LIN {X 0,Y 176.78,Z 239.076,A -85,B 0,C 180,E1 -23448.194,E2 -23448.194} C_VEL
LIN {X 0,Y 178.363,Z 246.541,A -85,B 0,C 180,E1 -23449.914,E2 -23449.914} C_VEL
LIN {X 0,Y 179.453,Z 256.138,A -85,B 0,C 180,E1 -23452.116,E2 -23452.116} C_VEL
LIN {X 0,Y 179.616,Z 266.645,A -85,B 0,C 180,E1 -23454.675,E2 -23454.675} C_VEL
LIN {X 0,Y 179.07,Z 275.287,A -85,B 0,C 180,E1 -23457.005,E2 -23457.005} C_VEL
LIN {X 0,Y 178.404,Z 280.467,A -85,B 0,C 180,E1 -23458.535,E2 -23458.535} C_VEL
LIN {X 0,Y 175.026,Z 289.302,A -85,B 0,C 180,E1 -23461.193,E2 -23461.193} C_VEL
LIN {X 0,Y 171.949,Z 296.845,A -85,B 0,C 180,E1 -23464.053,E2 -23464.053} C_VEL
LIN {X 0,Y 168.882,Z 303.785,A -85,B 0,C 180,E1 -23467.36,E2 -23467.36} C_VEL
LIN {X 0,Y 166.698,Z 308.639,A -85,B 0,C 180,E1 -23470.288,E2 -23470.288} C_VEL
LIN {X 0,Y 164.538,Z 313.357,A -85,B 0,C 180,E1 -23473.88,E2 -23473.88} C_VEL
LIN {X 0,Y 163.144,Z 316.97,A -85,B 0,C 180,E1 -23477.561,E2 -23477.561} C_VEL
LIN {X 0,Y 162.461,Z 318.833,A -85,B 0,C 180,E1 -23480.035,E2 -23480.035} C_VEL
LIN {X 0,Y 161.851,Z 321.235,A -85,B 0,C 180,E1 -23485.017,E2 -23485.017} C_VEL
LIN {X 0,Y 161.779,Z 321.876,A -85,B 0,C 180,E1 -23487.66,E2 -23487.66} C_VEL
LIN {X 0,Y 161.892,Z 322.064,A -85,B 0,C 180,E1 -23489.999,E2 -23489.999} C_VEL
LIN {X 0,Y 161.797,Z 321.836,A -85,B 0,C 180,E1 -23492.489,E2 -23492.489} C_VEL
LIN {X 0,Y 161.851,Z 321.217,A -85,B 0,C 180,E1 -23494.982,E2 -23494.982} C_VEL
LIN {X 0,Y 162.035,Z 320.208,A -85,B 0,C 180,E1 -23497.476,E2 -23497.476} C_VEL
LIN {X 0,Y 162.46,Z 318.797,A -85,B 0,C 180,E1 -23499.964,E2 -23499.964} C_VEL
LIN {X 0,Y 163.562,Z 315.842,A -85,B 0,C 180,E1 -23503.669,E2 -23503.669} C_VEL
LIN {X 0,Y 165.153,Z 311.848,A -85,B 0,C 180,E1 -23507.33,E2 -23507.33} C_VEL
LIN {X 0,Y 167.973,Z 305.719,A -85,B 0,C 180,E1 -23511.475,E2 -23511.475} C_VEL
LIN {X 0,Y 170.948,Z 299.153,A -85,B 0,C 180,E1 -23514.858,E2 -23514.858} C_VEL
LIN {X 0,Y 173.284,Z 293.389,A -85,B 0,C 180,E1 -23517.287,E2 -23517.287} C_VEL
LIN {X 0,Y 174.194,Z 289.612,A -85,B 0,C 180,E1 -23518.754,E2 -23518.754} C_VEL
LIN {X 0,Y 174.206,Z 285.779,A -85,B 0,C 180,E1 -23520.268,E2 -23520.268} C_VEL
LIN {X 0,Y 173.026,Z 275.11,A -85,B 0,C 180,E1 -23524.233,E2 -23524.233} C_VEL
LIN {X 0,Y 173.101,Z 272.13,A -85,B 0,C 180,E1 -23525.13,E2 -23525.13} C_VEL
LIN {X 0,Y 173.392,Z 261.231,A -85,B 0,C 180,E1 -23528.088,E2 -23528.088} C_VEL
LIN {X 0,Y 172.773,Z 251.105,A -85,B 0,C 180,E1 -23530.604,E2 -23530.604} C_VEL
LIN {X 0,Y 171.555,Z 243.424,A -85,B 0,C 180,E1 -23532.49,E2 -23532.49} C_VEL
LIN {X 0,Y 169.435,Z 236.666,A -85,B 0,C 180,E1 -23534.315,E2 -23534.315} C_VEL
LIN {X 0,Y 166.079,Z 229.215,A -85,B 0,C 180,E1 -23536.586,E2 -23536.586} C_VEL
LIN {X 0,Y 163.832,Z 224.747,A -85,B 0,C 180,E1 -23538.015,E2 -23538.015} C_VEL
LIN {X 0,Y 161.816,Z 220.984,A -85,B 0,C 180,E1 -23539.276,E2 -23539.276} C_VEL
LIN {X 0,Y 160.918,Z 219.536,A -85,B 0,C 180,E1 -23539.797,E2 -23539.797} C_VEL
LIN {X 0,Y 158.85,Z 216.171,A -85,B 0,C 180,E1 -23541.045,E2 -23541.045} C_VEL
LIN {X 0,Y 158.329,Z 214.418,A -85,B 0,C 180,E1 -23541.503,E2 -23541.503} C_VEL
LIN {X 0,Y 158.132,Z 212.84,A -85,B 0,C 180,E1 -23544.706,E2 -23544.706} C_VEL
LIN {X 0,Y 157.933,Z 211.437,A -85,B 0,C 180,E1 -23547.724,E2 -23547.724} C_VEL
LIN {X 0,Y 157.54,Z 209.207,A -85,B 0,C 180,E1 -23553.151,E2 -23553.151} C_VEL
LIN {X 0,Y 157.335,Z 208.061,A -85,B 0,C 180,E1 -23556.295,E2 -23556.295} C_VEL
LIN {X 0,Y 157.408,Z 207.878,A -85,B 0,C 180,E1 -23561.788,E2 -23561.788} C_VEL
LIN {X 0,Y 157.528,Z 207.864,A -85,B 0,C 180,E1 -23567.111,E2 -23567.111} C_VEL
LIN {X 0,Y 157.685,Z 207.834,A -85,B 0,C 180,E1 -23569.731,E2 -23569.731} C_VEL
LIN {X 0,Y 157.759,Z 207.833,A -85,B 0,C 180,E1 -23572.32,E2 -23572.32} C_VEL
LIN {X 0,Y 158.255,Z 207.772,A -85,B 0,C 180,E1 -23580,E2 -23580} C_VEL
LIN {X 0,Y 157.76,Z 207.832,A -85,B 0,C 180,E1 -23587.68,E2 -23587.68} C_VEL
LIN {X 0,Y 157.635,Z 207.85,A -85,B 0,C 180,E1 -23591.236,E2 -23591.236} C_VEL
LIN {X 0,Y 157.441,Z 207.871,A -85,B 0,C 180,E1 -23595.536,E2 -23595.536} C_VEL
LIN {X 0,Y 157.369,Z 207.88,A -85,B 0,C 180,E1 -23600.933,E2 -23600.933} C_VEL
LIN {X 0,Y 157.314,Z 207.89,A -85,B 0,C 180,E1 -23606.686,E2 -23606.686} C_VEL
LIN {X 0,Y 157.274,Z 207.896,A -85,B 0,C 180,E1 -23612.428,E2 -23612.428} C_VEL
LIN {X 0,Y 157.286,Z 207.969,A -85,B 0,C 180,E1 -23615.513,E2 -23615.513} C_VEL
LIN {X 0,Y 157.382,Z 209.037,A -85,B 0,C 180,E1 -23618.22,E2 -23618.22} C_VEL
LIN {X 0,Y 158.609,Z 211.909,A -85,B 0,C 180,E1 -23619.089,E2 -23619.089} C_VEL
LIN {X 0,Y 160.841,Z 214.656,A -85,B 0,C 180,E1 -23620.365,E2 -23620.365} C_VEL
LIN {X 0,Y 162.87,Z 218.288,A -85,B 0,C 180,E1 -23621.667,E2 -23621.667} C_VEL
LIN {X 0,Y 164.29,Z 220.876,A -85,B 0,C 180,E1 -23622.565,E2 -23622.565} C_VEL
LIN {X 0,Y 166.657,Z 225.258,A -85,B 0,C 180,E1 -23624.094,E2 -23624.094} C_VEL
LIN {X 0,Y 170.357,Z 233.531,A -85,B 0,C 180,E1 -23626.764,E2 -23626.764} C_VEL
LIN {X 0,Y 172.946,Z 242.042,A -85,B 0,C 180,E1 -23629.234,E2 -23629.234} C_VEL
LIN {X 0,Y 174.494,Z 250.978,A -85,B 0,C 180,E1 -23631.721,E2 -23631.721} C_VEL
LIN {X 0,Y 175.228,Z 260.194,A -85,B 0,C 180,E1 -23634.39,E2 -23634.39} C_VEL
LIN {X 0,Y 175.165,Z 267.085,A -85,B 0,C 180,E1 -23636.518,E2 -23636.518} C_VEL
LIN {X 0,Y 171.645,Z 276.507,A -85,B 0,C 180,E1 -23639.153,E2 -23639.153} C_VEL
LIN {X 0,Y 168.395,Z 284.517,A -85,B 0,C 180,E1 -23641.998,E2 -23641.998} C_VEL
LIN {X 0,Y 164.708,Z 292.19,A -85,B 0,C 180,E1 -23645.417,E2 -23645.417} C_VEL
LIN {X 0,Y 161.162,Z 299.236,A -85,B 0,C 180,E1 -23649.583,E2 -23649.583} C_VEL
LIN {X 0,Y 158.79,Z 303.922,A -85,B 0,C 180,E1 -23653.281,E2 -23653.281} C_VEL
LIN {X 0,Y 157.051,Z 307.504,A -85,B 0,C 180,E1 -23657.071,E2 -23657.071} C_VEL
LIN {X 0,Y 156.173,Z 309.352,A -85,B 0,C 180,E1 -23659.631,E2 -23659.631} C_VEL
LIN {X 0,Y 155.582,Z 310.738,A -85,B 0,C 180,E1 -23662.212,E2 -23662.212} C_VEL
LIN {X 0,Y 154.905,Z 312.331,A -85,B 0,C 180,E1 -23667.4,E2 -23667.4} C_VEL
LIN {X 0,Y 154.88,Z 312.556,A -85,B 0,C 180,E1 -23670.001,E2 -23670.001} C_VEL
LIN {X 0,Y 154.976,Z 312.124,A -85,B 0,C 180,E1 -23673.9,E2 -23673.9} C_VEL
LIN {X 0,Y 155.582,Z 310.806,A -85,B 0,C 180,E1 -23677.789,E2 -23677.789} C_VEL
LIN {X 0,Y 156.167,Z 309.45,A -85,B 0,C 180,E1 -23680.371,E2 -23680.371} C_VEL
LIN {X 0,Y 157.516,Z 306.582,A -85,B 0,C 180,E1 -23684.206,E2 -23684.206} C_VEL
LIN {X 0,Y 159.47,Z 302.69,A -85,B 0,C 180,E1 -23687.969,E2 -23687.969} C_VEL
LIN {X 0,Y 162.031,Z 297.666,A -85,B 0,C 180,E1 -23691.635,E2 -23691.635} C_VEL
LIN {X 0,Y 165.215,Z 291.334,A -85,B 0,C 180,E1 -23695.176,E2 -23695.176} C_VEL
LIN {X 0,Y 168.946,Z 283.412,A -85,B 0,C 180,E1 -23698.581,E2 -23698.581} C_VEL
LIN {X 0,Y 172.13,Z 275.519,A -85,B 0,C 180,E1 -23701.303,E2 -23701.303} C_VEL
LIN {X 0,Y 175.172,Z 267.617,A -85,B 0,C 180,E1 -23703.481,E2 -23703.481} C_VEL
LIN {X 0,Y 175.196,Z 258.051,A -85,B 0,C 180,E1 -23706.396,E2 -23706.396} C_VEL
LIN {X 0,Y 174.062,Z 247.419,A -85,B 0,C 180,E1 -23709.43,E2 -23709.43} C_VEL
LIN {X 0,Y 172.145,Z 238.94,A -85,B 0,C 180,E1 -23711.833,E2 -23711.833} C_VEL
LIN {X 0,Y 169.321,Z 230.807,A -85,B 0,C 180,E1 -23714.275,E2 -23714.275} C_VEL
LIN {X 0,Y 165.276,Z 222.609,A -85,B 0,C 180,E1 -23717.013,E2 -23717.013} C_VEL
LIN {X 0,Y 162.881,Z 218.324,A -85,B 0,C 180,E1 -23718.543,E2 -23718.543} C_VEL
LIN {X 0,Y 160.997,Z 214.957,A -85,B 0,C 180,E1 -23719.76,E2 -23719.76} C_VEL
LIN {X 0,Y 160.149,Z 213.715,A -85,B 0,C 180,E1 -23720.261,E2 -23720.261} C_VEL
LIN {X 0,Y 157.986,Z 210.749,A -85,B 0,C 180,E1 -23721.558,E2 -23721.558} C_VEL
LIN {X 0,Y 157.382,Z 208.874,A -85,B 0,C 180,E1 -23722.095,E2 -23722.095} C_VEL
LIN {X 0,Y 157.303,Z 208.062,A -85,B 0,C 180,E1 -23724.492,E2 -23724.492} C_VEL
LIN {X 0,Y 157.294,Z 207.888,A -85,B 0,C 180,E1 -23728.096,E2 -23728.096} C_VEL
LIN {X 0,Y 157.323,Z 207.883,A -85,B 0,C 180,E1 -23733.466,E2 -23733.466} C_VEL
LIN {X 0,Y 157.396,Z 207.879,A -85,B 0,C 180,E1 -23739.667,E2 -23739.667} C_VEL
LIN {X 0,Y 157.456,Z 207.872,A -85,B 0,C 180,E1 -23744.466,E2 -23744.466} C_VEL
LIN {X 0,Y 157.689,Z 207.842,A -85,B 0,C 180,E1 -23749.731,E2 -23749.731} C_VEL
LIN {X 0,Y 157.763,Z 207.832,A -85,B 0,C 180,E1 -23752.32,E2 -23752.32} C_VEL
LIN {X 0,Y 158.258,Z 207.77,A -85,B 0,C 180,E1 -23760,E2 -23760} C_VEL
LIN {X 0,Y 157.762,Z 207.834,A -85,B 0,C 180,E1 -23767.68,E2 -23767.68} C_VEL
LIN {X 0,Y 157.638,Z 207.852,A -85,B 0,C 180,E1 -23771.236,E2 -23771.236} C_VEL
LIN {X 0,Y 157.456,Z 207.875,A -85,B 0,C 180,E1 -23775.534,E2 -23775.534} C_VEL
LIN {X 0,Y 157.369,Z 207.883,A -85,B 0,C 180,E1 -23780.933,E2 -23780.933} C_VEL
LIN {X 0,Y 157.345,Z 208.125,A -85,B 0,C 180,E1 -23783.703,E2 -23783.703} C_VEL
LIN {X 0,Y 157.737,Z 210.255,A -85,B 0,C 180,E1 -23789.347,E2 -23789.347} C_VEL
LIN {X 0,Y 157.936,Z 211.5,A -85,B 0,C 180,E1 -23792.275,E2 -23792.275} C_VEL
LIN {X 0,Y 158.257,Z 213.7,A -85,B 0,C 180,E1 -23796.93,E2 -23796.93} C_VEL
LIN {X 0,Y 158.366,Z 214.446,A -85,B 0,C 180,E1 -23798.411,E2 -23798.411} C_VEL
LIN {X 0,Y 159.443,Z 217.379,A -85,B 0,C 180,E1 -23799.216,E2 -23799.216} C_VEL
LIN {X 0,Y 161.67,Z 220.578,A -85,B 0,C 180,E1 -23800.499,E2 -23800.499} C_VEL
LIN {X 0,Y 163.729,Z 224.606,A -85,B 0,C 180,E1 -23801.811,E2 -23801.811} C_VEL
LIN {X 0,Y 164.856,Z 226.613,A -85,B 0,C 180,E1 -23802.488,E2 -23802.488} C_VEL
LIN {X 0,Y 168.352,Z 233.944,A -85,B 0,C 180,E1 -23804.791,E2 -23804.791} C_VEL
LIN {X 0,Y 170.991,Z 241.181,A -85,B 0,C 180,E1 -23806.849,E2 -23806.849} C_VEL
LIN {X 0,Y 172.408,Z 247.523,A -85,B 0,C 180,E1 -23808.463,E2 -23808.463} C_VEL
LIN {X 0,Y 173.47,Z 258.738,A -85,B 0,C 180,E1 -23811.221,E2 -23811.221} C_VEL
LIN {X 0,Y 173.357,Z 268.826,A -85,B 0,C 180,E1 -23813.862,E2 -23813.862} C_VEL
LIN {X 0,Y 172.45,Z 278.275,A -85,B 0,C 180,E1 -23816.62,E2 -23816.62} C_VEL
LIN {X 0,Y 171.68,Z 282.204,A -85,B 0,C 180,E1 -23817.847,E2 -23817.847} C_VEL
LIN {X 0,Y 168.134,Z 290.669,A -85,B 0,C 180,E1 -23820.583,E2 -23820.583} C_VEL
LIN {X 0,Y 164.781,Z 298.441,A -85,B 0,C 180,E1 -23823.8,E2 -23823.8} C_VEL
LIN {X 0,Y 161.332,Z 305.608,A -85,B 0,C 180,E1 -23827.593,E2 -23827.593} C_VEL
LIN {X 0,Y 158.373,Z 311.709,A -85,B 0,C 180,E1 -23831.902,E2 -23831.902} C_VEL
LIN {X 0,Y 156.631,Z 315.682,A -85,B 0,C 180,E1 -23835.712,E2 -23835.712} C_VEL
LIN {X 0,Y 155.457,Z 318.62,A -85,B 0,C 180,E1 -23839.581,E2 -23839.581} C_VEL
LIN {X 0,Y 154.757,Z 321.022,A -85,B 0,C 180,E1 -23844.788,E2 -23844.788} C_VEL
LIN {X 0,Y 154.686,Z 321.748,A -85,B 0,C 180,E1 -23848.284,E2 -23848.284} C_VEL
LIN {X 0,Y 154.794,Z 321.851,A -85,B 0,C 180,E1 -23849.999,E2 -23849.999} C_VEL
LIN {X 0,Y 154.699,Z 321.623,A -85,B 0,C 180,E1 -23852.603,E2 -23852.603} C_VEL
LIN {X 0,Y 154.757,Z 321.003,A -85,B 0,C 180,E1 -23855.21,E2 -23855.21} C_VEL
LIN {X 0,Y 154.98,Z 319.994,A -85,B 0,C 180,E1 -23857.818,E2 -23857.818} C_VEL
LIN {X 0,Y 155.457,Z 318.583,A -85,B 0,C 180,E1 -23860.418,E2 -23860.418} C_VEL
LIN {X 0,Y 156.63,Z 315.627,A -85,B 0,C 180,E1 -23864.287,E2 -23864.287} C_VEL
LIN {X 0,Y 158.371,Z 311.633,A -85,B 0,C 180,E1 -23868.097,E2 -23868.097} C_VEL
LIN {X 0,Y 161.326,Z 305.502,A -85,B 0,C 180,E1 -23872.406,E2 -23872.406} C_VEL
LIN {X 0,Y 164.723,Z 298.399,A -85,B 0,C 180,E1 -23876.159,E2 -23876.159} C_VEL
LIN {X 0,Y 168.12,Z 290.511,A -85,B 0,C 180,E1 -23879.418,E2 -23879.418} C_VEL
LIN {X 0,Y 171.652,Z 282.002,A -85,B 0,C 180,E1 -23882.158,E2 -23882.158} C_VEL
LIN {X 0,Y 172.948,Z 273.749,A -85,B 0,C 180,E1 -23884.674,E2 -23884.674} C_VEL
LIN {X 0,Y 173.101,Z 272.13,A -85,B 0,C 180,E1 -23885.13,E2 -23885.13} C_VEL
LIN {X 0,Y 172.797,Z 267.849,A -85,B 0,C 180,E1 -23886.461,E2 -23886.461} C_VEL
LIN {X 0,Y 171.547,Z 263.857,A -85,B 0,C 180,E1 -23887.875,E2 -23887.875} C_VEL
LIN {X 0,Y 168.128,Z 256.123,A -85,B 0,C 180,E1 -23890.762,E2 -23890.762} C_VEL
LIN {X 0,Y 166.649,Z 250.286,A -85,B 0,C 180,E1 -23892.564,E2 -23892.564} C_VEL
LIN {X 0,Y 165.32,Z 243.61,A -85,B 0,C 180,E1 -23894.412,E2 -23894.412} C_VEL
LIN {X 0,Y 163.024,Z 237.373,A -85,B 0,C 180,E1 -23896.389,E2 -23896.389} C_VEL
LIN {X 0,Y 159.703,Z 229.94,A -85,B 0,C 180,E1 -23898.902,E2 -23898.902} C_VEL
LIN {X 0,Y 157.677,Z 225.941,A -85,B 0,C 180,E1 -23900.362,E2 -23900.362} C_VEL
LIN {X 0,Y 154.955,Z 221.098,A -85,B 0,C 180,E1 -23902.26,E2 -23902.26} C_VEL
LIN {X 0,Y 154.306,Z 219.798,A -85,B 0,C 180,E1 -23902.726,E2 -23902.726} C_VEL
LIN {X 0,Y 151.874,Z 216.371,A -85,B 0,C 180,E1 -23904.354,E2 -23904.354} C_VEL
LIN {X 0,Y 151.145,Z 214.074,A -85,B 0,C 180,E1 -23905.074,E2 -23905.074} C_VEL
LIN {X 0,Y 150.856,Z 212.313,A -85,B 0,C 180,E1 -23909.172,E2 -23909.172} C_VEL
LIN {X 0,Y 150.639,Z 211.045,A -85,B 0,C 180,E1 -23912.427,E2 -23912.427} C_VEL
LIN {X 0,Y 150.334,Z 209.112,A -85,B 0,C 180,E1 -23918.038,E2 -23918.038} C_VEL
LIN {X 0,Y 150.348,Z 208.759,A -85,B 0,C 180,E1 -23919.209,E2 -23919.209} C_VEL
LIN {X 0,Y 150.36,Z 208.755,A -85,B 0,C 180,E1 -23923.713,E2 -23923.713} C_VEL
LIN {X 0,Y 150.608,Z 208.714,A -85,B 0,C 180,E1 -23929.242,E2 -23929.242} C_VEL
LIN {X 0,Y 150.697,Z 208.714,A -85,B 0,C 180,E1 -23931.957,E2 -23931.957} C_VEL
LIN {X 0,Y 151.215,Z 208.65,A -85,B 0,C 180,E1 -23940,E2 -23940} C_VEL
LIN {X 0,Y 150.698,Z 208.713,A -85,B 0,C 180,E1 -23948.043,E2 -23948.043} C_VEL
LIN {X 0,Y 150.575,Z 208.729,A -85,B 0,C 180,E1 -23951.436,E2 -23951.436} C_VEL
LIN {X 0,Y 150.353,Z 208.755,A -85,B 0,C 180,E1 -23956.288,E2 -23956.288} C_VEL
LIN {X 0,Y 150.35,Z 208.754,A -85,B 0,C 180,E1 -23960.793,E2 -23960.793} C_VEL
LIN {X 0,Y 150.244,Z 208.769,A -85,B 0,C 180,E1 -23967.283,E2 -23967.283} C_VEL
LIN {X 0,Y 150.214,Z 208.775,A -85,B 0,C 180,E1 -23972.633,E2 -23972.633} C_VEL
LIN {X 0,Y 150.293,Z 209.416,A -85,B 0,C 180,E1 -23974.643,E2 -23974.643} C_VEL
LIN {X 0,Y 151.514,Z 212.159,A -85,B 0,C 180,E1 -23975.642,E2 -23975.642} C_VEL
LIN {X 0,Y 153.905,Z 215.12,A -85,B 0,C 180,E1 -23977.237,E2 -23977.237} C_VEL
LIN {X 0,Y 155.901,Z 218.643,A -85,B 0,C 180,E1 -23978.703,E2 -23978.703} C_VEL
LIN {X 0,Y 157.105,Z 220.386,A -85,B 0,C 180,E1 -23979.5,E2 -23979.5} C_VEL
LIN {X 0,Y 161.042,Z 227.816,A -85,B 0,C 180,E1 -23982.396,E2 -23982.396} C_VEL
LIN {X 0,Y 164.498,Z 235.616,A -85,B 0,C 180,E1 -23985.168,E2 -23985.168} C_VEL
LIN {X 0,Y 166.874,Z 243.25,A -85,B 0,C 180,E1 -23987.636,E2 -23987.636} C_VEL
LIN {X 0,Y 168.41,Z 252.094,A -85,B 0,C 180,E1 -23990.307,E2 -23990.307} C_VEL
LIN {X 0,Y 169.014,Z 261.573,A -85,B 0,C 180,E1 -23993.23,E2 -23993.23} C_VEL
LIN {X 0,Y 168.883,Z 268.368,A -85,B 0,C 180,E1 -23995.46,E2 -23995.46} C_VEL
LIN {X 0,Y 165.511,Z 276.891,A -85,B 0,C 180,E1 -23997.944,E2 -23997.944} C_VEL
LIN {X 0,Y 162.157,Z 284.733,A -85,B 0,C 180,E1 -24000.819,E2 -24000.819} C_VEL
LIN {X 0,Y 158.289,Z 292.405,A -85,B 0,C 180,E1 -24004.349,E2 -24004.349} C_VEL
LIN {X 0,Y 154.513,Z 299.451,A -85,B 0,C 180,E1 -24008.662,E2 -24008.662} C_VEL
LIN {X 0,Y 152.007,Z 304.137,A -85,B 0,C 180,E1 -24012.512,E2 -24012.512} C_VEL
LIN {X 0,Y 150.143,Z 307.718,A -85,B 0,C 180,E1 -24016.465,E2 -24016.465} C_VEL
LIN {X 0,Y 149.185,Z 309.567,A -85,B 0,C 180,E1 -24019.139,E2 -24019.139} C_VEL
LIN {X 0,Y 148.546,Z 310.952,A -85,B 0,C 180,E1 -24021.841,E2 -24021.841} C_VEL
LIN {X 0,Y 147.825,Z 312.544,A -85,B 0,C 180,E1 -24027.276,E2 -24027.276} C_VEL
LIN {X 0,Y 147.782,Z 312.769,A -85,B 0,C 180,E1 -24030.001,E2 -24030.001} C_VEL
LIN {X 0,Y 147.84,Z 312.467,A -85,B 0,C 180,E1 -24033.338,E2 -24033.338} C_VEL
LIN {X 0,Y 148.546,Z 311.019,A -85,B 0,C 180,E1 -24038.161,E2 -24038.161} C_VEL
LIN {X 0,Y 149.178,Z 309.663,A -85,B 0,C 180,E1 -24040.863,E2 -24040.863} C_VEL
LIN {X 0,Y 150.637,Z 306.795,A -85,B 0,C 180,E1 -24044.869,E2 -24044.869} C_VEL
LIN {X 0,Y 152.737,Z 302.902,A -85,B 0,C 180,E1 -24048.79,E2 -24048.79} C_VEL
LIN {X 0,Y 155.455,Z 297.878,A -85,B 0,C 180,E1 -24052.599,E2 -24052.599} C_VEL
LIN {X 0,Y 158.826,Z 291.545,A -85,B 0,C 180,E1 -24056.264,E2 -24056.264} C_VEL
LIN {X 0,Y 162.722,Z 283.659,A -85,B 0,C 180,E1 -24059.764,E2 -24059.764} C_VEL
LIN {X 0,Y 166.108,Z 275.729,A -85,B 0,C 180,E1 -24062.575,E2 -24062.575} C_VEL
LIN {X 0,Y 168.886,Z 268.892,A -85,B 0,C 180,E1 -24064.541,E2 -24064.541} C_VEL
LIN {X 0,Y 169.099,Z 260.842,A -85,B 0,C 180,E1 -24067.168,E2 -24067.168} C_VEL
LIN {X 0,Y 168.327,Z 250.867,A -85,B 0,C 180,E1 -24070.238,E2 -24070.238} C_VEL
LIN {X 0,Y 166.903,Z 243.346,A -85,B 0,C 180,E1 -24072.53,E2 -24072.53} C_VEL
LIN {X 0,Y 164.206,Z 234.837,A -85,B 0,C 180,E1 -24075.296,E2 -24075.296} C_VEL
LIN {X 0,Y 160.835,Z 227.437,A -85,B 0,C 180,E1 -24077.975,E2 -24077.975} C_VEL
LIN {X 0,Y 158.51,Z 223.061,A -85,B 0,C 180,E1 -24079.68,E2 -24079.68} C_VEL
LIN {X 0,Y 156.319,Z 219.085,A -85,B 0,C 180,E1 -24081.277,E2 -24081.277} C_VEL
LIN {X 0,Y 154.253,Z 215.867,A -85,B 0,C 180,E1 -24082.733,E2 -24082.733} C_VEL
LIN {X 0,Y 153.58,Z 214.548,A -85,B 0,C 180,E1 -24083.242,E2 -24083.242} C_VEL
LIN {X 0,Y 151.158,Z 211.637,A -85,B 0,C 180,E1 -24084.874,E2 -24084.874} C_VEL
LIN {X 0,Y 150.256,Z 209.221,A -85,B 0,C 180,E1 -24085.754,E2 -24085.754} C_VEL
LIN {X 0,Y 150.216,Z 208.77,A -85,B 0,C 180,E1 -24087.368,E2 -24087.368} C_VEL
LIN {X 0,Y 150.246,Z 208.769,A -85,B 0,C 180,E1 -24092.718,E2 -24092.718} C_VEL
LIN {X 0,Y 150.353,Z 208.754,A -85,B 0,C 180,E1 -24099.208,E2 -24099.208} C_VEL
LIN {X 0,Y 150.364,Z 208.753,A -85,B 0,C 180,E1 -24103.713,E2 -24103.713} C_VEL
LIN {X 0,Y 150.612,Z 208.725,A -85,B 0,C 180,E1 -24109.242,E2 -24109.242} C_VEL
LIN {X 0,Y 150.701,Z 208.713,A -85,B 0,C 180,E1 -24111.957,E2 -24111.957} C_VEL
LIN {X 0,Y 151.218,Z 208.647,A -85,B 0,C 180,E1 -24120,E2 -24120} C_VEL
LIN {X 0,Y 150.7,Z 208.715,A -85,B 0,C 180,E1 -24128.042,E2 -24128.042} C_VEL
LIN {X 0,Y 150.578,Z 208.731,A -85,B 0,C 180,E1 -24131.436,E2 -24131.436} C_VEL
LIN {X 0,Y 150.363,Z 208.756,A -85,B 0,C 180,E1 -24136.286,E2 -24136.286} C_VEL
LIN {X 0,Y 150.351,Z 208.793,A -85,B 0,C 180,E1 -24140.791,E2 -24140.791} C_VEL
LIN {X 0,Y 150.477,Z 210.129,A -85,B 0,C 180,E1 -24144.856,E2 -24144.856} C_VEL
LIN {X 0,Y 150.858,Z 212.378,A -85,B 0,C 180,E1 -24150.828,E2 -24150.828} C_VEL
LIN {X 0,Y 151.136,Z 214.092,A -85,B 0,C 180,E1 -24154.826,E2 -24154.826} C_VEL
LIN {X 0,Y 152.424,Z 217.416,A -85,B 0,C 180,E1 -24155.905,E2 -24155.905} C_VEL
LIN {X 0,Y 154.802,Z 220.594,A -85,B 0,C 180,E1 -24157.462,E2 -24157.462} C_VEL
LIN {X 0,Y 156.958,Z 224.728,A -85,B 0,C 180,E1 -24159.025,E2 -24159.025} C_VEL
LIN {X 0,Y 157.993,Z 226.704,A -85,B 0,C 180,E1 -24159.75,E2 -24159.75} C_VEL
LIN {X 0,Y 160.466,Z 231.532,A -85,B 0,C 180,E1 -24161.527,E2 -24161.527} C_VEL
LIN {X 0,Y 163.971,Z 239.709,A -85,B 0,C 180,E1 -24164.276,E2 -24164.276} C_VEL
LIN {X 0,Y 165.858,Z 245.626,A -85,B 0,C 180,E1 -24166.084,E2 -24166.084} C_VEL
LIN {X 0,Y 166.932,Z 252.193,A -85,B 0,C 180,E1 -24167.861,E2 -24167.861} C_VEL
LIN {X 0,Y 167.434,Z 261.38,A -85,B 0,C 180,E1 -24170.31,E2 -24170.31} C_VEL
LIN {X 0,Y 166.965,Z 272.479,A -85,B 0,C 180,E1 -24173.472,E2 -24173.472} C_VEL
LIN {X 0,Y 165.571,Z 281.989,A -85,B 0,C 180,E1 -24176.508,E2 -24176.508} C_VEL
LIN {X 0,Y 161.966,Z 290.458,A -85,B 0,C 180,E1 -24179.345,E2 -24179.345} C_VEL
LIN {X 0,Y 158.135,Z 298.799,A -85,B 0,C 180,E1 -24182.939,E2 -24182.939} C_VEL
LIN {X 0,Y 154.75,Z 305.396,A -85,B 0,C 180,E1 -24186.585,E2 -24186.585} C_VEL
LIN {X 0,Y 152.46,Z 309.907,A -85,B 0,C 180,E1 -24189.773,E2 -24189.773} C_VEL
LIN {X 0,Y 150.245,Z 314.242,A -85,B 0,C 180,E1 -24193.7,E2 -24193.7} C_VEL
LIN {X 0,Y 149.238,Z 316.544,A -85,B 0,C 180,E1 -24196.38,E2 -24196.38} C_VEL
LIN {X 0,Y 148.446,Z 318.407,A -85,B 0,C 180,E1 -24199.083,E2 -24199.083} C_VEL
LIN {X 0,Y 147.948,Z 319.807,A -85,B 0,C 180,E1 -24201.806,E2 -24201.806} C_VEL
LIN {X 0,Y 147.689,Z 320.809,A -85,B 0,C 180,E1 -24204.538,E2 -24204.538} C_VEL
LIN {X 0,Y 147.622,Z 321.571,A -85,B 0,C 180,E1 -24208.772,E2 -24208.772} C_VEL
LIN {X 0,Y 147.63,Z 321.559,A -85,B 0,C 180,E1 -24211.362,E2 -24211.362} C_VEL
LIN {X 0,Y 147.689,Z 320.79,A -85,B 0,C 180,E1 -24215.461,E2 -24215.461} C_VEL
LIN {X 0,Y 147.947,Z 319.78,A -85,B 0,C 180,E1 -24218.192,E2 -24218.192} C_VEL
LIN {X 0,Y 148.445,Z 318.368,A -85,B 0,C 180,E1 -24220.916,E2 -24220.916} C_VEL
LIN {X 0,Y 149.724,Z 315.412,A -85,B 0,C 180,E1 -24224.961,E2 -24224.961} C_VEL
LIN {X 0,Y 151.627,Z 311.418,A -85,B 0,C 180,E1 -24228.932,E2 -24228.932} C_VEL
LIN {X 0,Y 154.745,Z 305.286,A -85,B 0,C 180,E1 -24233.415,E2 -24233.415} C_VEL
LIN {X 0,Y 158.069,Z 298.764,A -85,B 0,C 180,E1 -24237.014,E2 -24237.014} C_VEL
LIN {X 0,Y 161.951,Z 290.294,A -85,B 0,C 180,E1 -24240.656,E2 -24240.656} C_VEL
LIN {X 0,Y 165.527,Z 281.78,A -85,B 0,C 180,E1 -24243.501,E2 -24243.501} C_VEL
LIN {X 0,Y 166.814,Z 273.519,A -85,B 0,C 180,E1 -24246.144,E2 -24246.144} C_VEL
LIN {X 0,Y 167.343,Z 263.534,A -85,B 0,C 180,E1 -24249.046,E2 -24249.046} C_VEL
LIN {X 0,Y 167.011,Z 253.718,A -85,B 0,C 180,E1 -24251.674,E2 -24251.674} C_VEL
LIN {X 0,Y 166.649,Z 250.286,A -85,B 0,C 180,E1 -24252.564,E2 -24252.564} C_VEL
LIN {X 0,Y 165.919,Z 247.414,A -85,B 0,C 180,E1 -24253.444,E2 -24253.444} C_VEL
LIN {X 0,Y 163.794,Z 243.883,A -85,B 0,C 180,E1 -24254.921,E2 -24254.921} C_VEL
LIN {X 0,Y 156.228,Z 236.19,A -85,B 0,C 180,E1 -24259.261,E2 -24259.261} C_VEL
LIN {X 0,Y 154.089,Z 232.501,A -85,B 0,C 180,E1 -24260.864,E2 -24260.864} C_VEL
LIN {X 0,Y 152.829,Z 229.787,A -85,B 0,C 180,E1 -24261.918,E2 -24261.918} C_VEL
LIN {X 0,Y 150.367,Z 225.002,A -85,B 0,C 180,E1 -24263.941,E2 -24263.941} C_VEL
LIN {X 0,Y 148.231,Z 221.395,A -85,B 0,C 180,E1 -24265.654,E2 -24265.654} C_VEL
LIN {X 0,Y 147.491,Z 219.75,A -85,B 0,C 180,E1 -24266.313,E2 -24266.313} C_VEL
LIN {X 0,Y 144.949,Z 216.601,A -85,B 0,C 180,E1 -24268.28,E2 -24268.28} C_VEL
LIN {X 0,Y 143.905,Z 213.739,A -85,B 0,C 180,E1 -24269.353,E2 -24269.353} C_VEL
LIN {X 0,Y 143.596,Z 212.105,A -85,B 0,C 180,E1 -24273.865,E2 -24273.865} C_VEL
LIN {X 0,Y 143.378,Z 210.166,A -85,B 0,C 180,E1 -24279.933,E2 -24279.933} C_VEL
LIN {X 0,Y 143.299,Z 209.637,A -85,B 0,C 180,E1 -24282.887,E2 -24282.887} C_VEL
LIN {X 0,Y 143.534,Z 209.596,A -85,B 0,C 180,E1 -24288.705,E2 -24288.705} C_VEL
LIN {X 0,Y 143.619,Z 209.596,A -85,B 0,C 180,E1 -24291.558,E2 -24291.558} C_VEL
LIN {X 0,Y 144.174,Z 209.527,A -85,B 0,C 180,E1 -24300,E2 -24300} C_VEL
LIN {X 0,Y 143.62,Z 209.596,A -85,B 0,C 180,E1 -24308.442,E2 -24308.442} C_VEL
LIN {X 0,Y 143.503,Z 209.611,A -85,B 0,C 180,E1 -24311.628,E2 -24311.628} C_VEL
LIN {X 0,Y 143.295,Z 209.636,A -85,B 0,C 180,E1 -24317.114,E2 -24317.114} C_VEL
LIN {X 0,Y 143.276,Z 209.636,A -85,B 0,C 180,E1 -24321.255,E2 -24321.255} C_VEL
LIN {X 0,Y 143.19,Z 209.648,A -85,B 0,C 180,E1 -24327.938,E2 -24327.938} C_VEL
LIN {X 0,Y 143.126,Z 209.669,A -85,B 0,C 180,E1 -24330.22,E2 -24330.22} C_VEL
LIN {X 0,Y 143.966,Z 212.152,A -85,B 0,C 180,E1 -24331.142,E2 -24331.142} C_VEL
LIN {X 0,Y 146.128,Z 214.662,A -85,B 0,C 180,E1 -24332.891,E2 -24332.891} C_VEL
LIN {X 0,Y 147.186,Z 215.737,A -85,B 0,C 180,E1 -24333.682,E2 -24333.682} C_VEL
LIN {X 0,Y 149.334,Z 219.458,A -85,B 0,C 180,E1 -24335.516,E2 -24335.516} C_VEL
LIN {X 0,Y 150.418,Z 221.069,A -85,B 0,C 180,E1 -24336.356,E2 -24336.356} C_VEL
LIN {X 0,Y 153.039,Z 225.54,A -85,B 0,C 180,E1 -24338.481,E2 -24338.481} C_VEL
LIN {X 0,Y 157.225,Z 234.245,A -85,B 0,C 180,E1 -24342.106,E2 -24342.106} C_VEL
LIN {X 0,Y 160.218,Z 242.319,A -85,B 0,C 180,E1 -24345.117,E2 -24345.117} C_VEL
LIN {X 0,Y 161.886,Z 249.48,A -85,B 0,C 180,E1 -24347.564,E2 -24347.564} C_VEL
LIN {X 0,Y 162.748,Z 257.87,A -85,B 0,C 180,E1 -24350.293,E2 -24350.293} C_VEL
LIN {X 0,Y 162.732,Z 267.548,A -85,B 0,C 180,E1 -24353.572,E2 -24353.572} C_VEL
LIN {X 0,Y 162.632,Z 269.639,A -85,B 0,C 180,E1 -24354.312,E2 -24354.312} C_VEL
LIN {X 0,Y 158.453,Z 279.514,A -85,B 0,C 180,E1 -24357.429,E2 -24357.429} C_VEL
LIN {X 0,Y 154.568,Z 287.679,A -85,B 0,C 180,E1 -24360.74,E2 -24360.74} C_VEL
LIN {X 0,Y 150.677,Z 294.84,A -85,B 0,C 180,E1 -24364.441,E2 -24364.441} C_VEL
LIN {X 0,Y 147.908,Z 299.666,A -85,B 0,C 180,E1 -24367.659,E2 -24367.659} C_VEL
LIN {X 0,Y 145.259,Z 304.351,A -85,B 0,C 180,E1 -24371.671,E2 -24371.671} C_VEL
LIN {X 0,Y 143.235,Z 307.932,A -85,B 0,C 180,E1 -24375.799,E2 -24375.799} C_VEL
LIN {X 0,Y 142.224,Z 309.78,A -85,B 0,C 180,E1 -24378.601,E2 -24378.601} C_VEL
LIN {X 0,Y 141.516,Z 311.166,A -85,B 0,C 180,E1 -24381.433,E2 -24381.433} C_VEL
LIN {X 0,Y 140.736,Z 312.757,A -85,B 0,C 180,E1 -24387.138,E2 -24387.138} C_VEL
LIN {X 0,Y 140.69,Z 312.982,A -85,B 0,C 180,E1 -24390.001,E2 -24390.001} C_VEL
LIN {X 0,Y 140.737,Z 312.786,A -85,B 0,C 180,E1 -24392.863,E2 -24392.863} C_VEL
LIN {X 0,Y 141.516,Z 311.231,A -85,B 0,C 180,E1 -24398.569,E2 -24398.569} C_VEL
LIN {X 0,Y 142.215,Z 309.875,A -85,B 0,C 180,E1 -24401.402,E2 -24401.402} C_VEL
LIN {X 0,Y 143.787,Z 307.007,A -85,B 0,C 180,E1 -24405.595,E2 -24405.595} C_VEL
LIN {X 0,Y 146.044,Z 303.113,A -85,B 0,C 180,E1 -24409.686,E2 -24409.686} C_VEL
LIN {X 0,Y 148.932,Z 298.089,A -85,B 0,C 180,E1 -24413.648,E2 -24413.648} C_VEL
LIN {X 0,Y 152.503,Z 291.755,A -85,B 0,C 180,E1 -24417.442,E2 -24417.442} C_VEL
LIN {X 0,Y 156.462,Z 284.114,A -85,B 0,C 180,E1 -24420.96,E2 -24420.96} C_VEL
LIN {X 0,Y 160.249,Z 275.763,A -85,B 0,C 180,E1 -24423.999,E2 -24423.999} C_VEL
LIN {X 0,Y 162.635,Z 270.119,A -85,B 0,C 180,E1 -24425.689,E2 -24425.689} C_VEL
LIN {X 0,Y 162.934,Z 262.161,A -85,B 0,C 180,E1 -24428.458,E2 -24428.458} C_VEL
LIN {X 0,Y 162.424,Z 252.944,A -85,B 0,C 180,E1 -24431.488,E2 -24431.488} C_VEL
LIN {X 0,Y 160.823,Z 244.33,A -85,B 0,C 180,E1 -24434.364,E2 -24434.364} C_VEL
LIN {X 0,Y 158.304,Z 236.737,A -85,B 0,C 180,E1 -24437.145,E2 -24437.145} C_VEL
LIN {X 0,Y 155.292,Z 230.006,A -85,B 0,C 180,E1 -24439.841,E2 -24439.841} C_VEL
LIN {X 0,Y 152.525,Z 224.635,A -85,B 0,C 180,E1 -24442.174,E2 -24442.174} C_VEL
LIN {X 0,Y 150.391,Z 220.874,A -85,B 0,C 180,E1 -24443.947,E2 -24443.947} C_VEL
LIN {X 0,Y 147.398,Z 216.312,A -85,B 0,C 180,E1 -24446.373,E2 -24446.373} C_VEL
LIN {X 0,Y 146.744,Z 215.08,A -85,B 0,C 180,E1 -24446.953,E2 -24446.953} C_VEL
LIN {X 0,Y 144.219,Z 212.591,A -85,B 0,C 180,E1 -24448.919,E2 -24448.919} C_VEL
LIN {X 0,Y 143.254,Z 210.347,A -85,B 0,C 180,E1 -24449.912,E2 -24449.912} C_VEL
LIN {X 0,Y 143.126,Z 209.652,A -85,B 0,C 180,E1 -24450.187,E2 -24450.187} C_VEL
LIN {X 0,Y 143.161,Z 209.646,A -85,B 0,C 180,E1 -24453.779,E2 -24453.779} C_VEL
LIN {X 0,Y 143.309,Z 209.635,A -85,B 0,C 180,E1 -24459.923,E2 -24459.923} C_VEL
LIN {X 0,Y 143.361,Z 209.626,A -85,B 0,C 180,E1 -24465.811,E2 -24465.811} C_VEL
LIN {X 0,Y 143.538,Z 209.605,A -85,B 0,C 180,E1 -24468.705,E2 -24468.705} C_VEL
LIN {X 0,Y 143.624,Z 209.596,A -85,B 0,C 180,E1 -24471.558,E2 -24471.558} C_VEL
LIN {X 0,Y 144.177,Z 209.524,A -85,B 0,C 180,E1 -24480,E2 -24480} C_VEL
LIN {X 0,Y 143.623,Z 209.598,A -85,B 0,C 180,E1 -24488.441,E2 -24488.441} C_VEL
LIN {X 0,Y 143.507,Z 209.611,A -85,B 0,C 180,E1 -24491.628,E2 -24491.628} C_VEL
LIN {X 0,Y 143.303,Z 209.637,A -85,B 0,C 180,E1 -24497.113,E2 -24497.113} C_VEL
LIN {X 0,Y 143.424,Z 210.617,A -85,B 0,C 180,E1 -24501.402,E2 -24501.402} C_VEL
LIN {X 0,Y 143.75,Z 212.945,A -85,B 0,C 180,E1 -24508.353,E2 -24508.353} C_VEL
LIN {X 0,Y 143.875,Z 213.754,A -85,B 0,C 180,E1 -24510.451,E2 -24510.451} C_VEL
LIN {X 0,Y 145.113,Z 216.902,A -85,B 0,C 180,E1 -24511.68,E2 -24511.68} C_VEL
LIN {X 0,Y 147.867,Z 220.374,A -85,B 0,C 180,E1 -24513.816,E2 -24513.816} C_VEL
LIN {X 0,Y 149.701,Z 224.109,A -85,B 0,C 180,E1 -24515.415,E2 -24515.415} C_VEL
LIN {X 0,Y 151.111,Z 226.22,A -85,B 0,C 180,E1 -24516.473,E2 -24516.473} C_VEL
LIN {X 0,Y 154.049,Z 232.273,A -85,B 0,C 180,E1 -24518.936,E2 -24518.936} C_VEL
LIN {X 0,Y 157.583,Z 240.151,A -85,B 0,C 180,E1 -24521.989,E2 -24521.989} C_VEL
LIN {X 0,Y 160.136,Z 247.746,A -85,B 0,C 180,E1 -24524.604,E2 -24524.604} C_VEL
LIN {X 0,Y 161.202,Z 254.533,A -85,B 0,C 180,E1 -24526.634,E2 -24526.634} C_VEL
LIN {X 0,Y 161.457,Z 263.622,A -85,B 0,C 180,E1 -24529.237,E2 -24529.237} C_VEL
LIN {X 0,Y 160.669,Z 274.35,A -85,B 0,C 180,E1 -24532.533,E2 -24532.533} C_VEL
LIN {X 0,Y 159.457,Z 281.77,A -85,B 0,C 180,E1 -24535.042,E2 -24535.042} C_VEL
LIN {X 0,Y 158.225,Z 285.366,A -85,B 0,C 180,E1 -24536.273,E2 -24536.273} C_VEL
LIN {X 0,Y 154.416,Z 293.226,A -85,B 0,C 180,E1 -24539.2,E2 -24539.2} C_VEL
LIN {X 0,Y 150.62,Z 300.913,A -85,B 0,C 180,E1 -24542.938,E2 -24542.938} C_VEL
LIN {X 0,Y 147.716,Z 306.178,A -85,B 0,C 180,E1 -24546.145,E2 -24546.145} C_VEL
LIN {X 0,Y 144.919,Z 311.285,A -85,B 0,C 180,E1 -24550.155,E2 -24550.155} C_VEL
LIN {X 0,Y 142.847,Z 315.255,A -85,B 0,C 180,E1 -24554.3,E2 -24554.3} C_VEL
LIN {X 0,Y 141.454,Z 318.194,A -85,B 0,C 180,E1 -24558.536,E2 -24558.536} C_VEL
LIN {X 0,Y 140.621,Z 320.596,A -85,B 0,C 180,E1 -24564.263,E2 -24564.263} C_VEL
LIN {X 0,Y 140.569,Z 321.396,A -85,B 0,C 180,E1 -24569.355,E2 -24569.355} C_VEL
LIN {X 0,Y 140.508,Z 321.196,A -85,B 0,C 180,E1 -24572.866,E2 -24572.866} C_VEL
LIN {X 0,Y 140.621,Z 320.576,A -85,B 0,C 180,E1 -24575.736,E2 -24575.736} C_VEL
LIN {X 0,Y 141.454,Z 318.153,A -85,B 0,C 180,E1 -24581.462,E2 -24581.462} C_VEL
LIN {X 0,Y 142.846,Z 315.197,A -85,B 0,C 180,E1 -24585.699,E2 -24585.699} C_VEL
LIN {X 0,Y 144.917,Z 311.204,A -85,B 0,C 180,E1 -24589.844,E2 -24589.844} C_VEL
LIN {X 0,Y 148.232,Z 305.071,A -85,B 0,C 180,E1 -24594.509,E2 -24594.509} C_VEL
LIN {X 0,Y 151.219,Z 299.619,A -85,B 0,C 180,E1 -24597.694,E2 -24597.694} C_VEL
LIN {X 0,Y 155.123,Z 291.569,A -85,B 0,C 180,E1 -24601.4,E2 -24601.4} C_VEL
LIN {X 0,Y 158.918,Z 283.372,A -85,B 0,C 180,E1 -24604.322,E2 -24604.322} C_VEL
LIN {X 0,Y 160.47,Z 275.457,A -85,B 0,C 180,E1 -24607.027,E2 -24607.027} C_VEL
LIN {X 0,Y 161.256,Z 265.952,A -85,B 0,C 180,E1 -24610.003,E2 -24610.003} C_VEL
LIN {X 0,Y 161.255,Z 256.764,A -85,B 0,C 180,E1 -24612.654,E2 -24612.654} C_VEL
LIN {X 0,Y 160.397,Z 249,A -85,B 0,C 180,E1 -24614.902,E2 -24614.902} C_VEL
LIN {X 0,Y 158.48,Z 242.594,A -85,B 0,C 180,E1 -24617.04,E2 -24617.04} C_VEL
LIN {X 0,Y 155.328,Z 234.932,A -85,B 0,C 180,E1 -24619.852,E2 -24619.852} C_VEL
LIN {X 0,Y 154.089,Z 232.501,A -85,B 0,C 180,E1 -24620.864,E2 -24620.864} C_VEL
LIN {X 0,Y 152.656,Z 230.282,A -85,B 0,C 180,E1 -24621.945,E2 -24621.945} C_VEL
LIN {X 0,Y 150.739,Z 228.859,A -85,B 0,C 180,E1 -24623.145,E2 -24623.145} C_VEL
LIN {X 0,Y 144.49,Z 225.853,A -85,B 0,C 180,E1 -24627.072,E2 -24627.072} C_VEL
LIN {X 0,Y 143.912,Z 225.321,A -85,B 0,C 180,E1 -24627.516,E2 -24627.516} C_VEL
LIN {X 0,Y 141.611,Z 221.881,A -85,B 0,C 180,E1 -24629.629,E2 -24629.629} C_VEL
LIN {X 0,Y 140.627,Z 219.645,A -85,B 0,C 180,E1 -24630.723,E2 -24630.723} C_VEL
LIN {X 0,Y 137.831,Z 216.42,A -85,B 0,C 180,E1 -24633.4,E2 -24633.4} C_VEL
LIN {X 0,Y 136.648,Z 213.533,A -85,B 0,C 180,E1 -24634.893,E2 -24634.893} C_VEL
LIN {X 0,Y 136.494,Z 212.112,A -85,B 0,C 180,E1 -24638.874,E2 -24638.874} C_VEL
LIN {X 0,Y 136.27,Z 210.583,A -85,B 0,C 180,E1 -24645.056,E2 -24645.056} C_VEL
LIN {X 0,Y 136.43,Z 210.483,A -85,B 0,C 180,E1 -24648.165,E2 -24648.165} C_VEL
LIN {X 0,Y 136.546,Z 210.474,A -85,B 0,C 180,E1 -24651.118,E2 -24651.118} C_VEL
LIN {X 0,Y 137.13,Z 210.404,A -85,B 0,C 180,E1 -24660,E2 -24660} C_VEL
LIN {X 0,Y 136.547,Z 210.476,A -85,B 0,C 180,E1 -24668.883,E2 -24668.883} C_VEL
LIN {X 0,Y 136.439,Z 210.489,A -85,B 0,C 180,E1 -24671.891,E2 -24671.891} C_VEL
LIN {X 0,Y 136.238,Z 210.512,A -85,B 0,C 180,E1 -24678.03,E2 -24678.03} C_VEL
LIN {X 0,Y 136.197,Z 210.519,A -85,B 0,C 180,E1 -24681.749,E2 -24681.749} C_VEL
LIN {X 0,Y 136.079,Z 210.549,A -85,B 0,C 180,E1 -24684.71,E2 -24684.71} C_VEL
LIN {X 0,Y 136.802,Z 212.857,A -85,B 0,C 180,E1 -24685.79,E2 -24685.79} C_VEL
LIN {X 0,Y 138.68,Z 215.139,A -85,B 0,C 180,E1 -24687.773,E2 -24687.773} C_VEL
LIN {X 0,Y 140.292,Z 216.322,A -85,B 0,C 180,E1 -24689.219,E2 -24689.219} C_VEL
LIN {X 0,Y 141.934,Z 219.521,A -85,B 0,C 180,E1 -24691.016,E2 -24691.016} C_VEL
LIN {X 0,Y 143.968,Z 221.825,A -85,B 0,C 180,E1 -24692.79,E2 -24692.79} C_VEL
LIN {X 0,Y 146.289,Z 225.758,A -85,B 0,C 180,E1 -24694.995,E2 -24694.995} C_VEL
LIN {X 0,Y 151.024,Z 235.382,A -85,B 0,C 180,E1 -24699.631,E2 -24699.631} C_VEL
LIN {X 0,Y 154.256,Z 243.797,A -85,B 0,C 180,E1 -24703.201,E2 -24703.201} C_VEL
LIN {X 0,Y 156.068,Z 251.514,A -85,B 0,C 180,E1 -24706.097,E2 -24706.097} C_VEL
LIN {X 0,Y 156.814,Z 260.397,A -85,B 0,C 180,E1 -24709.238,E2 -24709.238} C_VEL
LIN {X 0,Y 156.571,Z 268.833,A -85,B 0,C 180,E1 -24712.297,E2 -24712.297} C_VEL
LIN {X 0,Y 156.107,Z 271.806,A -85,B 0,C 180,E1 -24713.38,E2 -24713.38} C_VEL
LIN {X 0,Y 152.112,Z 280.621,A -85,B 0,C 180,E1 -24716.329,E2 -24716.329} C_VEL
LIN {X 0,Y 148.421,Z 287.894,A -85,B 0,C 180,E1 -24719.402,E2 -24719.402} C_VEL
LIN {X 0,Y 144.319,Z 295.055,A -85,B 0,C 180,E1 -24723.228,E2 -24723.228} C_VEL
LIN {X 0,Y 141.356,Z 299.881,A -85,B 0,C 180,E1 -24726.563,E2 -24726.563} C_VEL
LIN {X 0,Y 138.529,Z 304.565,A -85,B 0,C 180,E1 -24730.746,E2 -24730.746} C_VEL
LIN {X 0,Y 136.36,Z 308.146,A -85,B 0,C 180,E1 -24735.067,E2 -24735.067} C_VEL
LIN {X 0,Y 135.265,Z 309.994,A -85,B 0,C 180,E1 -24738.006,E2 -24738.006} C_VEL
LIN {X 0,Y 134.489,Z 311.38,A -85,B 0,C 180,E1 -24740.981,E2 -24740.981} C_VEL
LIN {X 0,Y 133.956,Z 312.365,A -85,B 0,C 180,E1 -24743.978,E2 -24743.978} C_VEL
LIN {X 0,Y 133.596,Z 313.105,A -85,B 0,C 180,E1 -24748.239,E2 -24748.239} C_VEL
LIN {X 0,Y 133.66,Z 312.998,A -85,B 0,C 180,E1 -24753.015,E2 -24753.015} C_VEL
LIN {X 0,Y 133.957,Z 312.412,A -85,B 0,C 180,E1 -24756.024,E2 -24756.024} C_VEL
LIN {X 0,Y 134.489,Z 311.444,A -85,B 0,C 180,E1 -24759.02,E2 -24759.02} C_VEL
LIN {X 0,Y 135.255,Z 310.088,A -85,B 0,C 180,E1 -24761.997,E2 -24761.997} C_VEL
LIN {X 0,Y 136.97,Z 307.219,A -85,B 0,C 180,E1 -24766.393,E2 -24766.393} C_VEL
LIN {X 0,Y 139.368,Z 303.325,A -85,B 0,C 180,E1 -24770.671,E2 -24770.671} C_VEL
LIN {X 0,Y 142.441,Z 298.301,A -85,B 0,C 180,E1 -24774.797,E2 -24774.797} C_VEL
LIN {X 0,Y 146.253,Z 291.966,A -85,B 0,C 180,E1 -24778.721,E2 -24778.721} C_VEL
LIN {X 0,Y 150.259,Z 284.605,A -85,B 0,C 180,E1 -24782.24,E2 -24782.24} C_VEL
LIN {X 0,Y 154.404,Z 275.972,A -85,B 0,C 180,E1 -24785.475,E2 -24785.475} C_VEL
LIN {X 0,Y 156.091,Z 272.271,A -85,B 0,C 180,E1 -24786.626,E2 -24786.626} C_VEL
LIN {X 0,Y 156.798,Z 267.235,A -85,B 0,C 180,E1 -24788.456,E2 -24788.456} C_VEL
LIN {X 0,Y 156.797,Z 258.768,A -85,B 0,C 180,E1 -24791.52,E2 -24791.52} C_VEL
LIN {X 0,Y 156.19,Z 251.913,A -85,B 0,C 180,E1 -24793.95,E2 -24793.95} C_VEL
LIN {X 0,Y 154.556,Z 244.591,A -85,B 0,C 180,E1 -24796.682,E2 -24796.682} C_VEL
LIN {X 0,Y 151.576,Z 236.579,A -85,B 0,C 180,E1 -24800.072,E2 -24800.072} C_VEL
LIN {X 0,Y 148.397,Z 229.785,A -85,B 0,C 180,E1 -24803.227,E2 -24803.227} C_VEL
LIN {X 0,Y 146.058,Z 225.476,A -85,B 0,C 180,E1 -24805.466,E2 -24805.466} C_VEL
LIN {X 0,Y 143.434,Z 220.983,A -85,B 0,C 180,E1 -24808.008,E2 -24808.008} C_VEL
LIN {X 0,Y 141.184,Z 218.334,A -85,B 0,C 180,E1 -24810.043,E2 -24810.043} C_VEL
LIN {X 0,Y 140.008,Z 216.018,A -85,B 0,C 180,E1 -24811.37,E2 -24811.37} C_VEL
LIN {X 0,Y 137.441,Z 213.817,A -85,B 0,C 180,E1 -24813.83,E2 -24813.83} C_VEL
LIN {X 0,Y 136.325,Z 211.646,A -85,B 0,C 180,E1 -24815.236,E2 -24815.236} C_VEL
LIN {X 0,Y 136.111,Z 210.531,A -85,B 0,C 180,E1 -24815.789,E2 -24815.789} C_VEL
LIN {X 0,Y 136.246,Z 210.508,A -85,B 0,C 180,E1 -24818.833,E2 -24818.833} C_VEL
LIN {X 0,Y 136.27,Z 210.51,A -85,B 0,C 180,E1 -24825.056,E2 -24825.056} C_VEL
LIN {X 0,Y 136.434,Z 210.489,A -85,B 0,C 180,E1 -24828.165,E2 -24828.165} C_VEL
LIN {X 0,Y 136.55,Z 210.475,A -85,B 0,C 180,E1 -24831.118,E2 -24831.118} C_VEL
LIN {X 0,Y 137.134,Z 210.401,A -85,B 0,C 180,E1 -24840,E2 -24840} C_VEL
LIN {X 0,Y 136.549,Z 210.479,A -85,B 0,C 180,E1 -24848.882,E2 -24848.882} C_VEL
LIN {X 0,Y 136.442,Z 210.491,A -85,B 0,C 180,E1 -24851.89,E2 -24851.89} C_VEL
LIN {X 0,Y 136.302,Z 210.649,A -85,B 0,C 180,E1 -24854.94,E2 -24854.94} C_VEL
LIN {X 0,Y 136.501,Z 212.167,A -85,B 0,C 180,E1 -24861.125,E2 -24861.125} C_VEL
LIN {X 0,Y 136.553,Z 213.266,A -85,B 0,C 180,E1 -24864.719,E2 -24864.719} C_VEL
LIN {X 0,Y 137.863,Z 216.449,A -85,B 0,C 180,E1 -24866.389,E2 -24866.389} C_VEL
LIN {X 0,Y 140.609,Z 219.621,A -85,B 0,C 180,E1 -24869.047,E2 -24869.047} C_VEL
LIN {X 0,Y 142.964,Z 224.14,A -85,B 0,C 180,E1 -24871.488,E2 -24871.488} C_VEL
LIN {X 0,Y 144.433,Z 226.172,A -85,B 0,C 180,E1 -24872.775,E2 -24872.775} C_VEL
LIN {X 0,Y 146.438,Z 230.193,A -85,B 0,C 180,E1 -24874.744,E2 -24874.744} C_VEL
LIN {X 0,Y 150.316,Z 238.646,A -85,B 0,C 180,E1 -24878.535,E2 -24878.535} C_VEL
LIN {X 0,Y 153.294,Z 246.297,A -85,B 0,C 180,E1 -24881.665,E2 -24881.665} C_VEL
LIN {X 0,Y 155.077,Z 253.094,A -85,B 0,C 180,E1 -24884.123,E2 -24884.123} C_VEL
LIN {X 0,Y 155.559,Z 259.989,A -85,B 0,C 180,E1 -24886.291,E2 -24886.291} C_VEL
LIN {X 0,Y 155.271,Z 268.602,A -85,B 0,C 180,E1 -24888.98,E2 -24888.98} C_VEL
LIN {X 0,Y 154.122,Z 277.982,A -85,B 0,C 180,E1 -24892.159,E2 -24892.159} C_VEL
LIN {X 0,Y 152.965,Z 283.359,A -85,B 0,C 180,E1 -24894.14,E2 -24894.14} C_VEL
LIN {X 0,Y 150.694,Z 288.458,A -85,B 0,C 180,E1 -24895.968,E2 -24895.968} C_VEL
LIN {X 0,Y 146.889,Z 295.751,A -85,B 0,C 180,E1 -24899.047,E2 -24899.047} C_VEL
LIN {X 0,Y 143.066,Z 302.939,A -85,B 0,C 180,E1 -24902.973,E2 -24902.973} C_VEL
LIN {X 0,Y 140.178,Z 307.789,A -85,B 0,C 180,E1 -24906.353,E2 -24906.353} C_VEL
LIN {X 0,Y 137.379,Z 312.506,A -85,B 0,C 180,E1 -24910.577,E2 -24910.577} C_VEL
LIN {X 0,Y 135.418,Z 316.117,A -85,B 0,C 180,E1 -24914.959,E2 -24914.959} C_VEL
LIN {X 0,Y 134.487,Z 317.981,A -85,B 0,C 180,E1 -24917.934,E2 -24917.934} C_VEL
LIN {X 0,Y 133.547,Z 320.383,A -85,B 0,C 180,E1 -24923.958,E2 -24923.958} C_VEL
LIN {X 0,Y 133.411,Z 320.995,A -85,B 0,C 180,E1 -24926.98,E2 -24926.98} C_VEL
LIN {X 0,Y 133.532,Z 321.213,A -85,B 0,C 180,E1 -24929.999,E2 -24929.999} C_VEL
LIN {X 0,Y 133.411,Z 320.982,A -85,B 0,C 180,E1 -24933.019,E2 -24933.019} C_VEL
LIN {X 0,Y 133.547,Z 320.363,A -85,B 0,C 180,E1 -24936.041,E2 -24936.041} C_VEL
LIN {X 0,Y 134.486,Z 317.939,A -85,B 0,C 180,E1 -24942.065,E2 -24942.065} C_VEL
LIN {X 0,Y 135.974,Z 314.981,A -85,B 0,C 180,E1 -24946.515,E2 -24946.515} C_VEL
LIN {X 0,Y 138.223,Z 310.988,A -85,B 0,C 180,E1 -24950.849,E2 -24950.849} C_VEL
LIN {X 0,Y 141.789,Z 304.855,A -85,B 0,C 180,E1 -24955.702,E2 -24955.702} C_VEL
LIN {X 0,Y 145.401,Z 298.412,A -85,B 0,C 180,E1 -24959.537,E2 -24959.537} C_VEL
LIN {X 0,Y 149.861,Z 289.861,A -85,B 0,C 180,E1 -24963.437,E2 -24963.437} C_VEL
LIN {X 0,Y 152.926,Z 283.149,A -85,B 0,C 180,E1 -24965.869,E2 -24965.869} C_VEL
LIN {X 0,Y 154.483,Z 275.143,A -85,B 0,C 180,E1 -24968.753,E2 -24968.753} C_VEL
LIN {X 0,Y 155.356,Z 265.71,A -85,B 0,C 180,E1 -24971.855,E2 -24971.855} C_VEL
LIN {X 0,Y 155.39,Z 256.884,A -85,B 0,C 180,E1 -24974.575,E2 -24974.575} C_VEL
LIN {X 0,Y 154.769,Z 251.609,A -85,B 0,C 180,E1 -24976.263,E2 -24976.263} C_VEL
LIN {X 0,Y 153.19,Z 246.093,A -85,B 0,C 180,E1 -24978.3,E2 -24978.3} C_VEL
LIN {X 0,Y 149.713,Z 237.302,A -85,B 0,C 180,E1 -24981.907,E2 -24981.907} C_VEL
LIN {X 0,Y 146.096,Z 229.71,A -85,B 0,C 180,E1 -24985.372,E2 -24985.372} C_VEL
LIN {X 0,Y 143.912,Z 225.321,A -85,B 0,C 180,E1 -24987.516,E2 -24987.516} C_VEL
LIN {X 0,Y 140.582,Z 222.656,A -85,B 0,C 180,E1 -24990.192,E2 -24990.192} C_VEL
LIN {X 0,Y 132.785,Z 218.351,A -85,B 0,C 180,E1 -24997.642,E2 -24997.642} C_VEL
LIN {X 0,Y 131.574,Z 217.186,A -85,B 0,C 180,E1 -24999.203,E2 -24999.203} C_VEL
LIN {X 0,Y 129.854,Z 214.124,A -85,B 0,C 180,E1 -25002.072,E2 -25002.072} C_VEL
LIN {X 0,Y 129.398,Z 212.686,A -85,B 0,C 180,E1 -25003.23,E2 -25003.23} C_VEL
LIN {X 0,Y 129.413,Z 211.72,A -85,B 0,C 180,E1 -25007.824,E2 -25007.824} C_VEL
LIN {X 0,Y 129.47,Z 211.351,A -85,B 0,C 180,E1 -25010.628,E2 -25010.628} C_VEL
LIN {X 0,Y 130.085,Z 211.281,A -85,B 0,C 180,E1 -25020,E2 -25020} C_VEL
LIN {X 0,Y 129.47,Z 211.355,A -85,B 0,C 180,E1 -25029.372,E2 -25029.372} C_VEL
LIN {X 0,Y 129.342,Z 211.371,A -85,B 0,C 180,E1 -25032.553,E2 -25032.553} C_VEL
LIN {X 0,Y 129.201,Z 211.565,A -85,B 0,C 180,E1 -25037.001,E2 -25037.001} C_VEL
LIN {X 0,Y 130.07,Z 214.097,A -85,B 0,C 180,E1 -25038.917,E2 -25038.917} C_VEL
LIN {X 0,Y 132.68,Z 216.729,A -85,B 0,C 180,E1 -25042.619,E2 -25042.619} C_VEL
LIN {X 0,Y 133.614,Z 217.389,A -85,B 0,C 180,E1 -25043.748,E2 -25043.748} C_VEL
LIN {X 0,Y 135.048,Z 220.367,A -85,B 0,C 180,E1 -25045.839,E2 -25045.839} C_VEL
LIN {X 0,Y 137.365,Z 222.711,A -85,B 0,C 180,E1 -25048.35,E2 -25048.35} C_VEL
LIN {X 0,Y 139.026,Z 225.798,A -85,B 0,C 180,E1 -25050.366,E2 -25050.366} C_VEL
LIN {X 0,Y 140.373,Z 227.293,A -85,B 0,C 180,E1 -25051.667,E2 -25051.667} C_VEL
LIN {X 0,Y 144.38,Z 235.398,A -85,B 0,C 180,E1 -25056.246,E2 -25056.246} C_VEL
LIN {X 0,Y 147.646,Z 243.346,A -85,B 0,C 180,E1 -25060.165,E2 -25060.165} C_VEL
LIN {X 0,Y 149.546,Z 249.792,A -85,B 0,C 180,E1 -25063.005,E2 -25063.005} C_VEL
LIN {X 0,Y 150.643,Z 256.241,A -85,B 0,C 180,E1 -25065.59,E2 -25065.59} C_VEL
LIN {X 0,Y 150.832,Z 264.501,A -85,B 0,C 180,E1 -25068.733,E2 -25068.733} C_VEL
LIN {X 0,Y 150.24,Z 272.031,A -85,B 0,C 180,E1 -25071.698,E2 -25071.698} C_VEL
LIN {X 0,Y 147.895,Z 277.536,A -85,B 0,C 180,E1 -25073.56,E2 -25073.56} C_VEL
LIN {X 0,Y 143.756,Z 285.67,A -85,B 0,C 180,E1 -25076.801,E2 -25076.801} C_VEL
LIN {X 0,Y 139.382,Z 293.051,A -85,B 0,C 180,E1 -25080.554,E2 -25080.554} C_VEL
LIN {X 0,Y 134.861,Z 300.096,A -85,B 0,C 180,E1 -25085.362,E2 -25085.362} C_VEL
LIN {X 0,Y 131.848,Z 304.78,A -85,B 0,C 180,E1 -25089.729,E2 -25089.729} C_VEL
LIN {X 0,Y 129.52,Z 308.36,A -85,B 0,C 180,E1 -25094.259,E2 -25094.259} C_VEL
LIN {X 0,Y 128.316,Z 310.209,A -85,B 0,C 180,E1 -25097.346,E2 -25097.346} C_VEL
LIN {X 0,Y 127.492,Z 311.593,A -85,B 0,C 180,E1 -25100.482,E2 -25100.482} C_VEL
LIN {X 0,Y 126.585,Z 313.183,A -85,B 0,C 180,E1 -25106.818,E2 -25106.818} C_VEL
LIN {X 0,Y 126.505,Z 313.407,A -85,B 0,C 180,E1 -25110.001,E2 -25110.001} C_VEL
LIN {X 0,Y 126.585,Z 313.211,A -85,B 0,C 180,E1 -25113.183,E2 -25113.183} C_VEL
LIN {X 0,Y 127.491,Z 311.657,A -85,B 0,C 180,E1 -25119.52,E2 -25119.52} C_VEL
LIN {X 0,Y 128.306,Z 310.3,A -85,B 0,C 180,E1 -25122.657,E2 -25122.657} C_VEL
LIN {X 0,Y 130.169,Z 307.431,A -85,B 0,C 180,E1 -25127.275,E2 -25127.275} C_VEL
LIN {X 0,Y 132.743,Z 303.537,A -85,B 0,C 180,E1 -25131.754,E2 -25131.754} C_VEL
LIN {X 0,Y 136.018,Z 298.513,A -85,B 0,C 180,E1 -25136.053,E2 -25136.053} C_VEL
LIN {X 0,Y 140.068,Z 292.177,A -85,B 0,C 180,E1 -25140.117,E2 -25140.117} C_VEL
LIN {X 0,Y 144.016,Z 285.336,A -85,B 0,C 180,E1 -25143.525,E2 -25143.525} C_VEL
LIN {X 0,Y 148.668,Z 276.182,A -85,B 0,C 180,E1 -25147.066,E2 -25147.066} C_VEL
LIN {X 0,Y 150.262,Z 272.487,A -85,B 0,C 180,E1 -25148.297,E2 -25148.297} C_VEL
LIN {X 0,Y 150.913,Z 265.033,A -85,B 0,C 180,E1 -25151.246,E2 -25151.246} C_VEL
LIN {X 0,Y 150.687,Z 256.092,A -85,B 0,C 180,E1 -25154.663,E2 -25154.663} C_VEL
LIN {X 0,Y 149.455,Z 249.084,A -85,B 0,C 180,E1 -25157.49,E2 -25157.49} C_VEL
LIN {X 0,Y 147.23,Z 242.027,A -85,B 0,C 180,E1 -25160.677,E2 -25160.677} C_VEL
LIN {X 0,Y 144.236,Z 234.966,A -85,B 0,C 180,E1 -25164.217,E2 -25164.217} C_VEL
LIN {X 0,Y 140.132,Z 226.953,A -85,B 0,C 180,E1 -25168.887,E2 -25168.887} C_VEL
LIN {X 0,Y 138.041,Z 224.199,A -85,B 0,C 180,E1 -25171.075,E2 -25171.075} C_VEL
LIN {X 0,Y 137.095,Z 222.269,A -85,B 0,C 180,E1 -25172.317,E2 -25172.317} C_VEL
LIN {X 0,Y 134.738,Z 219.89,A -85,B 0,C 180,E1 -25174.925,E2 -25174.925} C_VEL
LIN {X 0,Y 133.569,Z 217.144,A -85,B 0,C 180,E1 -25176.757,E2 -25176.757} C_VEL
LIN {X 0,Y 130.554,Z 214.815,A -85,B 0,C 180,E1 -25180.748,E2 -25180.748} C_VEL
LIN {X 0,Y 129.269,Z 212.008,A -85,B 0,C 180,E1 -25183.314,E2 -25183.314} C_VEL
LIN {X 0,Y 129.179,Z 211.391,A -85,B 0,C 180,E1 -25183.81,E2 -25183.81} C_VEL
LIN {X 0,Y 129.392,Z 211.366,A -85,B 0,C 180,E1 -25187.875,E2 -25187.875} C_VEL
LIN {X 0,Y 129.474,Z 211.355,A -85,B 0,C 180,E1 -25190.628,E2 -25190.628} C_VEL
LIN {X 0,Y 130.088,Z 211.279,A -85,B 0,C 180,E1 -25200,E2 -25200} C_VEL
LIN {X 0,Y 129.473,Z 211.359,A -85,B 0,C 180,E1 -25209.372,E2 -25209.372} C_VEL
LIN {X 0,Y 129.418,Z 211.866,A -85,B 0,C 180,E1 -25212.546,E2 -25212.546} C_VEL
LIN {X 0,Y 129.45,Z 212.889,A -85,B 0,C 180,E1 -25216.662,E2 -25216.662} C_VEL
LIN {X 0,Y 130.998,Z 216.4,A -85,B 0,C 180,E1 -25219.591,E2 -25219.591} C_VEL
LIN {X 0,Y 134.101,Z 219.868,A -85,B 0,C 180,E1 -25223.7,E2 -25223.7} C_VEL
LIN {X 0,Y 135.949,Z 223.764,A -85,B 0,C 180,E1 -25226.273,E2 -25226.273} C_VEL
LIN {X 0,Y 137.867,Z 226.162,A -85,B 0,C 180,E1 -25228.341,E2 -25228.341} C_VEL
LIN {X 0,Y 139.521,Z 229.751,A -85,B 0,C 180,E1 -25230.391,E2 -25230.391} C_VEL
LIN {X 0,Y 140.338,Z 230.899,A -85,B 0,C 180,E1 -25231.203,E2 -25231.203} C_VEL
LIN {X 0,Y 143.697,Z 238.278,A -85,B 0,C 180,E1 -25235.077,E2 -25235.077} C_VEL
LIN {X 0,Y 147.188,Z 247.245,A -85,B 0,C 180,E1 -25239.248,E2 -25239.248} C_VEL
LIN {X 0,Y 149.399,Z 255.145,A -85,B 0,C 180,E1 -25242.535,E2 -25242.535} C_VEL
LIN {X 0,Y 149.82,Z 261.462,A -85,B 0,C 180,E1 -25244.72,E2 -25244.72} C_VEL
LIN {X 0,Y 149.222,Z 270.869,A -85,B 0,C 180,E1 -25247.887,E2 -25247.887} C_VEL
LIN {X 0,Y 147.792,Z 279.818,A -85,B 0,C 180,E1 -25251.144,E2 -25251.144} C_VEL
LIN {X 0,Y 146.463,Z 284.939,A -85,B 0,C 180,E1 -25253.143,E2 -25253.143} C_VEL
LIN {X 0,Y 142.356,Z 292.803,A -85,B 0,C 180,E1 -25256.261,E2 -25256.261} C_VEL
LIN {X 0,Y 138.343,Z 299.97,A -85,B 0,C 180,E1 -25259.923,E2 -25259.923} C_VEL
LIN {X 0,Y 134.786,Z 305.753,A -85,B 0,C 180,E1 -25263.691,E2 -25263.691} C_VEL
LIN {X 0,Y 131.585,Z 310.859,A -85,B 0,C 180,E1 -25268.045,E2 -25268.045} C_VEL
LIN {X 0,Y 129.146,Z 314.828,A -85,B 0,C 180,E1 -25272.583,E2 -25272.583} C_VEL
LIN {X 0,Y 127.515,Z 317.767,A -85,B 0,C 180,E1 -25277.263,E2 -25277.263} C_VEL
LIN {X 0,Y 126.469,Z 320.17,A -85,B 0,C 180,E1 -25283.618,E2 -25283.618} C_VEL
LIN {X 0,Y 126.314,Z 320.782,A -85,B 0,C 180,E1 -25286.81,E2 -25286.81} C_VEL
LIN {X 0,Y 126.445,Z 321,A -85,B 0,C 180,E1 -25289.999,E2 -25289.999} C_VEL
LIN {X 0,Y 126.314,Z 320.769,A -85,B 0,C 180,E1 -25293.189,E2 -25293.189} C_VEL
LIN {X 0,Y 126.468,Z 320.148,A -85,B 0,C 180,E1 -25296.38,E2 -25296.38} C_VEL
LIN {X 0,Y 127.514,Z 317.724,A -85,B 0,C 180,E1 -25302.735,E2 -25302.735} C_VEL
LIN {X 0,Y 129.145,Z 314.766,A -85,B 0,C 180,E1 -25307.415,E2 -25307.415} C_VEL
LIN {X 0,Y 131.583,Z 310.773,A -85,B 0,C 180,E1 -25311.954,E2 -25311.954} C_VEL
LIN {X 0,Y 135.42,Z 304.64,A -85,B 0,C 180,E1 -25317.006,E2 -25317.006} C_VEL
LIN {X 0,Y 138.875,Z 298.82,A -85,B 0,C 180,E1 -25320.648,E2 -25320.648} C_VEL
LIN {X 0,Y 143.137,Z 291.136,A -85,B 0,C 180,E1 -25324.377,E2 -25324.377} C_VEL
LIN {X 0,Y 146.424,Z 284.724,A -85,B 0,C 180,E1 -25326.867,E2 -25326.867} C_VEL
LIN {X 0,Y 148.075,Z 278.1,A -85,B 0,C 180,E1 -25329.422,E2 -25329.422} C_VEL
LIN {X 0,Y 149.371,Z 268.402,A -85,B 0,C 180,E1 -25332.892,E2 -25332.892} C_VEL
LIN {X 0,Y 149.739,Z 259.67,A -85,B 0,C 180,E1 -25335.782,E2 -25335.782} C_VEL
LIN {X 0,Y 149.29,Z 254.855,A -85,B 0,C 180,E1 -25337.472,E2 -25337.472} C_VEL
LIN {X 0,Y 147.745,Z 248.961,A -85,B 0,C 180,E1 -25339.868,E2 -25339.868} C_VEL
LIN {X 0,Y 144.89,Z 241.139,A -85,B 0,C 180,E1 -25343.377,E2 -25343.377} C_VEL
LIN {X 0,Y 142.355,Z 235.313,A -85,B 0,C 180,E1 -25346.261,E2 -25346.261} C_VEL
LIN {X 0,Y 139.842,Z 230.263,A -85,B 0,C 180,E1 -25349.07,E2 -25349.07} C_VEL
LIN {X 0,Y 137.906,Z 226.363,A -85,B 0,C 180,E1 -25351.356,E2 -25351.356} C_VEL
LIN {X 0,Y 136.709,Z 224.741,A -85,B 0,C 180,E1 -25352.648,E2 -25352.648} C_VEL
LIN {X 0,Y 134.606,Z 221.31,A -85,B 0,C 180,E1 -25355.208,E2 -25355.208} C_VEL
LIN {X 0,Y 133.856,Z 219.523,A -85,B 0,C 180,E1 -25356.328,E2 -25356.328} C_VEL
LIN {X 0,Y 131.574,Z 217.186,A -85,B 0,C 180,E1 -25359.203,E2 -25359.203} C_VEL
LIN {X 0,Y 129.837,Z 215.902,A -85,B 0,C 180,E1 -25361.62,E2 -25361.62} C_VEL
LIN {X 0,Y 127.022,Z 215.753,A -85,B 0,C 180,E1 -25365.873,E2 -25365.873} C_VEL
LIN {X 0,Y 124.47,Z 216.173,A -85,B 0,C 180,E1 -25371.257,E2 -25371.257} C_VEL
LIN {X 0,Y 123.965,Z 215.836,A -85,B 0,C 180,E1 -25373.09,E2 -25373.09} C_VEL
LIN {X 0,Y 123.392,Z 213.656,A -85,B 0,C 180,E1 -25380,E2 -25380} C_VEL
LIN {X 0,Y 127.204,Z 218.434,A -85,B 0,C 180,E1 -25396.14,E2 -25396.14} C_VEL
LIN {X 0,Y 128.408,Z 221.361,A -85,B 0,C 180,E1 -25398.964,E2 -25398.964} C_VEL
LIN {X 0,Y 130.994,Z 223.892,A -85,B 0,C 180,E1 -25402.891,E2 -25402.891} C_VEL
LIN {X 0,Y 132.351,Z 226.718,A -85,B 0,C 180,E1 -25405.139,E2 -25405.139} C_VEL
LIN {X 0,Y 134.554,Z 229.736,A -85,B 0,C 180,E1 -25408.04,E2 -25408.04} C_VEL
LIN {X 0,Y 136.862,Z 233.3,A -85,B 0,C 180,E1 -25410.898,E2 -25410.898} C_VEL
LIN {X 0,Y 140.052,Z 240.433,A -85,B 0,C 180,E1 -25415.246,E2 -25415.246} C_VEL
LIN {X 0,Y 142.593,Z 247.348,A -85,B 0,C 180,E1 -25418.933,E2 -25418.933} C_VEL
LIN {X 0,Y 144.148,Z 253.233,A -85,B 0,C 180,E1 -25421.78,E2 -25421.78} C_VEL
LIN {X 0,Y 144.994,Z 259.8,A -85,B 0,C 180,E1 -25424.653,E2 -25424.653} C_VEL
LIN {X 0,Y 144.847,Z 267.327,A -85,B 0,C 180,E1 -25427.739,E2 -25427.739} C_VEL
LIN {X 0,Y 144.379,Z 272.262,A -85,B 0,C 180,E1 -25429.837,E2 -25429.837} C_VEL
LIN {X 0,Y 143.947,Z 274.184,A -85,B 0,C 180,E1 -25430.603,E2 -25430.603} C_VEL
LIN {X 0,Y 139.212,Z 283.399,A -85,B 0,C 180,E1 -25434.076,E2 -25434.076} C_VEL
LIN {X 0,Y 134.821,Z 290.875,A -85,B 0,C 180,E1 -25437.703,E2 -25437.703} C_VEL
LIN {X 0,Y 131.096,Z 296.509,A -85,B 0,C 180,E1 -25441.153,E2 -25441.153} C_VEL
LIN {X 0,Y 127.303,Z 301.997,A -85,B 0,C 180,E1 -25445.541,E2 -25445.541} C_VEL
LIN {X 0,Y 124.285,Z 306.299,A -85,B 0,C 180,E1 -25450.168,E2 -25450.168} C_VEL
LIN {X 0,Y 122.683,Z 308.575,A -85,B 0,C 180,E1 -25453.357,E2 -25453.357} C_VEL
LIN {X 0,Y 121.401,Z 310.422,A -85,B 0,C 180,E1 -25456.612,E2 -25456.612} C_VEL
LIN {X 0,Y 120.49,Z 311.807,A -85,B 0,C 180,E1 -25459.923,E2 -25459.923} C_VEL
LIN {X 0,Y 119.498,Z 313.396,A -85,B 0,C 180,E1 -25466.629,E2 -25466.629} C_VEL
LIN {X 0,Y 119.419,Z 313.62,A -85,B 0,C 180,E1 -25470.001,E2 -25470.001} C_VEL
LIN {X 0,Y 119.499,Z 313.424,A -85,B 0,C 180,E1 -25473.372,E2 -25473.372} C_VEL
LIN {X 0,Y 120.489,Z 311.869,A -85,B 0,C 180,E1 -25480.079,E2 -25480.079} C_VEL
LIN {X 0,Y 121.388,Z 310.513,A -85,B 0,C 180,E1 -25483.391,E2 -25483.391} C_VEL
LIN {X 0,Y 123.389,Z 307.644,A -85,B 0,C 180,E1 -25488.257,E2 -25488.257} C_VEL
LIN {X 0,Y 126.175,Z 303.749,A -85,B 0,C 180,E1 -25492.949,E2 -25492.949} C_VEL
LIN {X 0,Y 129.673,Z 298.725,A -85,B 0,C 180,E1 -25497.432,E2 -25497.432} C_VEL
LIN {X 0,Y 133.968,Z 292.388,A -85,B 0,C 180,E1 -25501.642,E2 -25501.642} C_VEL
LIN {X 0,Y 138.911,Z 284.181,A -85,B 0,C 180,E1 -25505.752,E2 -25505.752} C_VEL
LIN {X 0,Y 143.937,Z 274.617,A -85,B 0,C 180,E1 -25509.402,E2 -25509.402} C_VEL
LIN {X 0,Y 144.638,Z 270.796,A -85,B 0,C 180,E1 -25510.994,E2 -25510.994} C_VEL
LIN {X 0,Y 145.148,Z 261.448,A -85,B 0,C 180,E1 -25514.87,E2 -25514.87} C_VEL
LIN {X 0,Y 144.701,Z 256.061,A -85,B 0,C 180,E1 -25517.159,E2 -25517.159} C_VEL
LIN {X 0,Y 143.524,Z 250.55,A -85,B 0,C 180,E1 -25519.718,E2 -25519.718} C_VEL
LIN {X 0,Y 141.891,Z 245.159,A -85,B 0,C 180,E1 -25522.42,E2 -25522.42} C_VEL
LIN {X 0,Y 139.192,Z 238.306,A -85,B 0,C 180,E1 -25526.261,E2 -25526.261} C_VEL
LIN {X 0,Y 137.041,Z 233.736,A -85,B 0,C 180,E1 -25529.146,E2 -25529.146} C_VEL
LIN {X 0,Y 134.232,Z 228.773,A -85,B 0,C 180,E1 -25532.883,E2 -25532.883} C_VEL
LIN {X 0,Y 131.726,Z 225.604,A -85,B 0,C 180,E1 -25536.204,E2 -25536.204} C_VEL
LIN {X 0,Y 130.774,Z 223.497,A -85,B 0,C 180,E1 -25537.902,E2 -25537.902} C_VEL
LIN {X 0,Y 128.354,Z 221.252,A -85,B 0,C 180,E1 -25541.649,E2 -25541.649} C_VEL
LIN {X 0,Y 127.08,Z 218.152,A -85,B 0,C 180,E1 -25544.77,E2 -25544.77} C_VEL
LIN {X 0,Y 123.607,Z 214.177,A -85,B 0,C 180,E1 -25560,E2 -25560} C_VEL
LIN {X 0,Y 125.275,Z 217.307,A -85,B 0,C 180,E1 -25570.625,E2 -25570.625} C_VEL
LIN {X 0,Y 127.531,Z 219.649,A -85,B 0,C 180,E1 -25575.789,E2 -25575.789} C_VEL
LIN {X 0,Y 129.011,Z 223.172,A -85,B 0,C 180,E1 -25579.078,E2 -25579.078} C_VEL
LIN {X 0,Y 131.4,Z 226.197,A -85,B 0,C 180,E1 -25582.712,E2 -25582.712} C_VEL
LIN {X 0,Y 132.794,Z 229.498,A -85,B 0,C 180,E1 -25585.049,E2 -25585.049} C_VEL
LIN {X 0,Y 134.635,Z 232.317,A -85,B 0,C 180,E1 -25587.45,E2 -25587.45} C_VEL
LIN {X 0,Y 137.482,Z 238.63,A -85,B 0,C 180,E1 -25591.407,E2 -25591.407} C_VEL
LIN {X 0,Y 140.246,Z 245.462,A -85,B 0,C 180,E1 -25595.19,E2 -25595.19} C_VEL
LIN {X 0,Y 142.709,Z 253.035,A -85,B 0,C 180,E1 -25598.894,E2 -25598.894} C_VEL
LIN {X 0,Y 143.976,Z 258.786,A -85,B 0,C 180,E1 -25601.446,E2 -25601.446} C_VEL
LIN {X 0,Y 144.054,Z 264.958,A -85,B 0,C 180,E1 -25603.746,E2 -25603.746} C_VEL
LIN {X 0,Y 143.021,Z 274.142,A -85,B 0,C 180,E1 -25607.101,E2 -25607.101} C_VEL
LIN {X 0,Y 141.154,Z 282.918,A -85,B 0,C 180,E1 -25610.593,E2 -25610.593} C_VEL
LIN {X 0,Y 139.976,Z 286.401,A -85,B 0,C 180,E1 -25612.043,E2 -25612.043} C_VEL
LIN {X 0,Y 134.845,Z 295.326,A -85,B 0,C 180,E1 -25615.924,E2 -25615.924} C_VEL
LIN {X 0,Y 130.834,Z 301.995,A -85,B 0,C 180,E1 -25619.789,E2 -25619.789} C_VEL
LIN {X 0,Y 127.204,Z 307.363,A -85,B 0,C 180,E1 -25623.768,E2 -25623.768} C_VEL
LIN {X 0,Y 124.019,Z 312.081,A -85,B 0,C 180,E1 -25628.386,E2 -25628.386} C_VEL
LIN {X 0,Y 121.699,Z 315.691,A -85,B 0,C 180,E1 -25633.216,E2 -25633.216} C_VEL
LIN {X 0,Y 120.575,Z 317.554,A -85,B 0,C 180,E1 -25636.517,E2 -25636.517} C_VEL
LIN {X 0,Y 119.415,Z 319.957,A -85,B 0,C 180,E1 -25643.239,E2 -25643.239} C_VEL
LIN {X 0,Y 119.228,Z 320.569,A -85,B 0,C 180,E1 -25646.62,E2 -25646.62} C_VEL
LIN {X 0,Y 119.36,Z 320.787,A -85,B 0,C 180,E1 -25649.999,E2 -25649.999} C_VEL
LIN {X 0,Y 119.415,Z 319.935,A -85,B 0,C 180,E1 -25656.759,E2 -25656.759} C_VEL
LIN {X 0,Y 120.574,Z 317.51,A -85,B 0,C 180,E1 -25663.482,E2 -25663.482} C_VEL
LIN {X 0,Y 122.358,Z 314.551,A -85,B 0,C 180,E1 -25668.415,E2 -25668.415} C_VEL
LIN {X 0,Y 125.002,Z 310.558,A -85,B 0,C 180,E1 -25673.175,E2 -25673.175} C_VEL
LIN {X 0,Y 129.133,Z 304.426,A -85,B 0,C 180,E1 -25678.437,E2 -25678.437} C_VEL
LIN {X 0,Y 133.326,Z 297.73,A -85,B 0,C 180,E1 -25682.703,E2 -25682.703} C_VEL
LIN {X 0,Y 138.191,Z 289.429,A -85,B 0,C 180,E1 -25686.695,E2 -25686.695} C_VEL
LIN {X 0,Y 139.94,Z 286.199,A -85,B 0,C 180,E1 -25687.966,E2 -25687.966} C_VEL
LIN {X 0,Y 141.894,Z 279.65,A -85,B 0,C 180,E1 -25690.658,E2 -25690.658} C_VEL
LIN {X 0,Y 143.411,Z 270.727,A -85,B 0,C 180,E1 -25694.087,E2 -25694.087} C_VEL
LIN {X 0,Y 144.089,Z 262.56,A -85,B 0,C 180,E1 -25697.022,E2 -25697.022} C_VEL
LIN {X 0,Y 143.87,Z 258.391,A -85,B 0,C 180,E1 -25698.607,E2 -25698.607} C_VEL
LIN {X 0,Y 142.102,Z 251.276,A -85,B 0,C 180,E1 -25701.816,E2 -25701.816} C_VEL
LIN {X 0,Y 139.097,Z 242.483,A -85,B 0,C 180,E1 -25706.235,E2 -25706.235} C_VEL
LIN {X 0,Y 136.434,Z 236.17,A -85,B 0,C 180,E1 -25709.852,E2 -25709.852} C_VEL
LIN {X 0,Y 134.247,Z 231.515,A -85,B 0,C 180,E1 -25712.867,E2 -25712.867} C_VEL
LIN {X 0,Y 131.952,Z 227.871,A -85,B 0,C 180,E1 -25715.934,E2 -25715.934} C_VEL
LIN {X 0,Y 131.032,Z 225.658,A -85,B 0,C 180,E1 -25717.533,E2 -25717.533} C_VEL
LIN {X 0,Y 128.115,Z 221.572,A -85,B 0,C 180,E1 -25722.233,E2 -25722.233} C_VEL
LIN {X 0,Y 127.328,Z 219.313,A -85,B 0,C 180,E1 -25724.185,E2 -25724.185} C_VEL
LIN {X 0,Y 124.262,Z 216.186,A -85,B 0,C 180,E1 -25731.872,E2 -25731.872} C_VEL
LIN {X 0,Y 123.965,Z 215.836,A -85,B 0,C 180,E1 -25733.09,E2 -25733.09} C_VEL
LIN {X 0,Y 123.562,Z 215.69,A -85,B 0,C 180,E1 -25734.903,E2 -25734.903} C_VEL
LIN {X 0,Y 123.162,Z 216.191,A -85,B 0,C 180,E1 -25736.714,E2 -25736.714} C_VEL
LIN {X 0,Y 122.466,Z 218.384,A -85,B 0,C 180,E1 -25740.281,E2 -25740.281} C_VEL
LIN {X 0,Y 122.089,Z 222.147,A -85,B 0,C 180,E1 -25745.714,E2 -25745.714} C_VEL
LIN {X 0,Y 122.353,Z 222.816,A -85,B 0,C 180,E1 -25747.58,E2 -25747.58} C_VEL
LIN {X 0,Y 124.961,Z 225.14,A -85,B 0,C 180,E1 -25755.39,E2 -25755.39} C_VEL
LIN {X 0,Y 125.822,Z 227.545,A -85,B 0,C 180,E1 -25757.893,E2 -25757.893} C_VEL
LIN {X 0,Y 127.471,Z 229.563,A -85,B 0,C 180,E1 -25761.001,E2 -25761.001} C_VEL
LIN {X 0,Y 128.33,Z 230.869,A -85,B 0,C 180,E1 -25762.542,E2 -25762.542} C_VEL
LIN {X 0,Y 131.449,Z 236.29,A -85,B 0,C 180,E1 -25767.698,E2 -25767.698} C_VEL
LIN {X 0,Y 133.112,Z 239.105,A -85,B 0,C 180,E1 -25770.105,E2 -25770.105} C_VEL
LIN {X 0,Y 135.866,Z 246.117,A -85,B 0,C 180,E1 -25774.681,E2 -25774.681} C_VEL
LIN {X 0,Y 137.929,Z 252.974,A -85,B 0,C 180,E1 -25778.569,E2 -25778.569} C_VEL
LIN {X 0,Y 139.06,Z 259.175,A -85,B 0,C 180,E1 -25781.738,E2 -25781.738} C_VEL
LIN {X 0,Y 139.252,Z 265.07,A -85,B 0,C 180,E1 -25784.441,E2 -25784.441} C_VEL
LIN {X 0,Y 138.518,Z 272.765,A -85,B 0,C 180,E1 -25787.896,E2 -25787.896} C_VEL
LIN {X 0,Y 138.281,Z 274.411,A -85,B 0,C 180,E1 -25788.647,E2 -25788.647} C_VEL
LIN {X 0,Y 136.728,Z 277.968,A -85,B 0,C 180,E1 -25790.022,E2 -25790.022} C_VEL
LIN {X 0,Y 132.26,Z 285.716,A -85,B 0,C 180,E1 -25793.225,E2 -25793.225} C_VEL
LIN {X 0,Y 128.027,Z 292.317,A -85,B 0,C 180,E1 -25796.706,E2 -25796.706} C_VEL
LIN {X 0,Y 123.468,Z 298.72,A -85,B 0,C 180,E1 -25801.065,E2 -25801.065} C_VEL
LIN {X 0,Y 119.728,Z 303.793,A -85,B 0,C 180,E1 -25805.74,E2 -25805.74} C_VEL
LIN {X 0,Y 116.689,Z 307.732,A -85,B 0,C 180,E1 -25810.656,E2 -25810.656} C_VEL
LIN {X 0,Y 114.516,Z 310.636,A -85,B 0,C 180,E1 -25815.79,E2 -25815.79} C_VEL
LIN {X 0,Y 113.518,Z 312.02,A -85,B 0,C 180,E1 -25819.297,E2 -25819.297} C_VEL
LIN {X 0,Y 112.425,Z 313.609,A -85,B 0,C 180,E1 -25826.417,E2 -25826.417} C_VEL
LIN {X 0,Y 112.335,Z 313.833,A -85,B 0,C 180,E1 -25830.001,E2 -25830.001} C_VEL
LIN {X 0,Y 112.425,Z 313.636,A -85,B 0,C 180,E1 -25833.585,E2 -25833.585} C_VEL
LIN {X 0,Y 113.516,Z 312.082,A -85,B 0,C 180,E1 -25840.705,E2 -25840.705} C_VEL
LIN {X 0,Y 114.503,Z 310.725,A -85,B 0,C 180,E1 -25844.213,E2 -25844.213} C_VEL
LIN {X 0,Y 116.65,Z 307.857,A -85,B 0,C 180,E1 -25849.353,E2 -25849.353} C_VEL
LIN {X 0,Y 119.649,Z 303.962,A -85,B 0,C 180,E1 -25854.279,E2 -25854.279} C_VEL
LIN {X 0,Y 123.415,Z 298.936,A -85,B 0,C 180,E1 -25858.95,E2 -25858.95} C_VEL
LIN {X 0,Y 127.975,Z 292.599,A -85,B 0,C 180,E1 -25863.311,E2 -25863.311} C_VEL
LIN {X 0,Y 132.896,Z 284.91,A -85,B 0,C 180,E1 -25867.307,E2 -25867.307} C_VEL
LIN {X 0,Y 137.599,Z 276.603,A -85,B 0,C 180,E1 -25870.634,E2 -25870.634} C_VEL
LIN {X 0,Y 138.29,Z 274.836,A -85,B 0,C 180,E1 -25871.352,E2 -25871.352} C_VEL
LIN {X 0,Y 139.273,Z 266.671,A -85,B 0,C 180,E1 -25875.051,E2 -25875.051} C_VEL
LIN {X 0,Y 139.307,Z 260.923,A -85,B 0,C 180,E1 -25877.643,E2 -25877.643} C_VEL
LIN {X 0,Y 138.418,Z 254.986,A -85,B 0,C 180,E1 -25880.595,E2 -25880.595} C_VEL
LIN {X 0,Y 136.893,Z 249.107,A -85,B 0,C 180,E1 -25883.814,E2 -25883.814} C_VEL
LIN {X 0,Y 134.739,Z 242.945,A -85,B 0,C 180,E1 -25887.592,E2 -25887.592} C_VEL
LIN {X 0,Y 133.294,Z 239.477,A -85,B 0,C 180,E1 -25889.941,E2 -25889.941} C_VEL
LIN {X 0,Y 130.982,Z 235.033,A -85,B 0,C 180,E1 -25893.555,E2 -25893.555} C_VEL
LIN {X 0,Y 129.375,Z 232.928,A -85,B 0,C 180,E1 -25895.957,E2 -25895.957} C_VEL
LIN {X 0,Y 128.543,Z 231.254,A -85,B 0,C 180,E1 -25897.497,E2 -25897.497} C_VEL
LIN {X 0,Y 126.834,Z 228.898,A -85,B 0,C 180,E1 -25900.581,E2 -25900.581} C_VEL
LIN {X 0,Y 125.392,Z 226.459,A -85,B 0,C 180,E1 -25903.83,E2 -25903.83} C_VEL
LIN {X 0,Y 124.973,Z 224.907,A -85,B 0,C 180,E1 -25905.341,E2 -25905.341} C_VEL
LIN {X 0,Y 122.112,Z 221.198,A -85,B 0,C 180,E1 -25920,E2 -25920} C_VEL
LIN {X 0,Y 123.648,Z 224.294,A -85,B 0,C 180,E1 -25930.645,E2 -25930.645} C_VEL
LIN {X 0,Y 125.28,Z 226.234,A -85,B 0,C 180,E1 -25934.934,E2 -25934.934} C_VEL
LIN {X 0,Y 126.795,Z 229.996,A -85,B 0,C 180,E1 -25938.794,E2 -25938.794} C_VEL
LIN {X 0,Y 128.227,Z 231.87,A -85,B 0,C 180,E1 -25941.289,E2 -25941.289} C_VEL
LIN {X 0,Y 129.57,Z 235.344,A -85,B 0,C 180,E1 -25944.004,E2 -25944.004} C_VEL
LIN {X 0,Y 131.02,Z 237.81,A -85,B 0,C 180,E1 -25946.254,E2 -25946.254} C_VEL
LIN {X 0,Y 133.277,Z 243.398,A -85,B 0,C 180,E1 -25950.063,E2 -25950.063} C_VEL
LIN {X 0,Y 135.545,Z 249.889,A -85,B 0,C 180,E1 -25953.942,E2 -25953.942} C_VEL
LIN {X 0,Y 137.786,Z 258.173,A -85,B 0,C 180,E1 -25958.307,E2 -25958.307} C_VEL
LIN {X 0,Y 138.527,Z 262.67,A -85,B 0,C 180,E1 -25960.446,E2 -25960.446} C_VEL
LIN {X 0,Y 138.284,Z 268.163,A -85,B 0,C 180,E1 -25962.644,E2 -25962.644} C_VEL
LIN {X 0,Y 136.945,Z 276.504,A -85,B 0,C 180,E1 -25965.929,E2 -25965.929} C_VEL
LIN {X 0,Y 134.893,Z 284.501,A -85,B 0,C 180,E1 -25969.363,E2 -25969.363} C_VEL
LIN {X 0,Y 133.512,Z 287.824,A -85,B 0,C 180,E1 -25970.825,E2 -25970.825} C_VEL
LIN {X 0,Y 128.985,Z 295.113,A -85,B 0,C 180,E1 -25974.144,E2 -25974.144} C_VEL
LIN {X 0,Y 124.517,Z 302.081,A -85,B 0,C 180,E1 -25978.335,E2 -25978.335} C_VEL
LIN {X 0,Y 120.842,Z 307.15,A -85,B 0,C 180,E1 -25982.272,E2 -25982.272} C_VEL
LIN {X 0,Y 117.428,Z 311.868,A -85,B 0,C 180,E1 -25987.105,E2 -25987.105} C_VEL
LIN {X 0,Y 114.871,Z 315.477,A -85,B 0,C 180,E1 -25992.186,E2 -25992.186} C_VEL
LIN {X 0,Y 113.665,Z 317.341,A -85,B 0,C 180,E1 -25995.68,E2 -25995.68} C_VEL
LIN {X 0,Y 112.34,Z 319.744,A -85,B 0,C 180,E1 -26002.811,E2 -26002.811} C_VEL
LIN {X 0,Y 112.137,Z 320.356,A -85,B 0,C 180,E1 -26006.406,E2 -26006.406} C_VEL
LIN {X 0,Y 112.261,Z 320.574,A -85,B 0,C 180,E1 -26009.999,E2 -26009.999} C_VEL
LIN {X 0,Y 112.137,Z 320.342,A -85,B 0,C 180,E1 -26013.592,E2 -26013.592} C_VEL
LIN {X 0,Y 112.34,Z 319.721,A -85,B 0,C 180,E1 -26017.187,E2 -26017.187} C_VEL
LIN {X 0,Y 113.664,Z 317.295,A -85,B 0,C 180,E1 -26024.318,E2 -26024.318} C_VEL
LIN {X 0,Y 115.597,Z 314.336,A -85,B 0,C 180,E1 -26029.534,E2 -26029.534} C_VEL
LIN {X 0,Y 118.488,Z 310.343,A -85,B 0,C 180,E1 -26034.531,E2 -26034.531} C_VEL
LIN {X 0,Y 122.936,Z 304.211,A -85,B 0,C 180,E1 -26040.013,E2 -26040.013} C_VEL
LIN {X 0,Y 127.371,Z 297.513,A -85,B 0,C 180,E1 -26044.441,E2 -26044.441} C_VEL
LIN {X 0,Y 132.542,Z 289.212,A -85,B 0,C 180,E1 -26048.537,E2 -26048.537} C_VEL
LIN {X 0,Y 134.251,Z 285.977,A -85,B 0,C 180,E1 -26049.887,E2 -26049.887} C_VEL
LIN {X 0,Y 136.206,Z 279.369,A -85,B 0,C 180,E1 -26052.771,E2 -26052.771} C_VEL
LIN {X 0,Y 137.83,Z 270.854,A -85,B 0,C 180,E1 -26056.216,E2 -26056.216} C_VEL
LIN {X 0,Y 138.5,Z 263.071,A -85,B 0,C 180,E1 -26059.254,E2 -26059.254} C_VEL
LIN {X 0,Y 137.824,Z 258.63,A -85,B 0,C 180,E1 -26061.334,E2 -26061.334} C_VEL
LIN {X 0,Y 135.806,Z 251.035,A -85,B 0,C 180,E1 -26065.302,E2 -26065.302} C_VEL
LIN {X 0,Y 133.567,Z 244.44,A -85,B 0,C 180,E1 -26069.135,E2 -26069.135} C_VEL
LIN {X 0,Y 132.726,Z 241.912,A -85,B 0,C 180,E1 -26070.673,E2 -26070.673} C_VEL
LIN {X 0,Y 130.388,Z 236.709,A -85,B 0,C 180,E1 -26074.456,E2 -26074.456} C_VEL
LIN {X 0,Y 127.774,Z 231.454,A -85,B 0,C 180,E1 -26079.054,E2 -26079.054} C_VEL
LIN {X 0,Y 125.494,Z 227.313,A -85,B 0,C 180,E1 -26083.739,E2 -26083.739} C_VEL
LIN {X 0,Y 125.149,Z 225.912,A -85,B 0,C 180,E1 -26084.946,E2 -26084.946} C_VEL
LIN {X 0,Y 122.517,Z 222.964,A -85,B 0,C 180,E1 -26092.584,E2 -26092.584} C_VEL
LIN {X 0,Y 121.909,Z 220.728,A -85,B 0,C 180,E1 -26100,E2 -26100} C_VEL
LIN {X 0,Y 122.353,Z 222.816,A -85,B 0,C 180,E1 -26107.58,E2 -26107.58} C_VEL
LIN {X 0,Y 122.61,Z 223.836,A -85,B 0,C 180,E1 -26109.349,E2 -26109.349} C_VEL
LIN {X 0,Y 122.66,Z 225.736,A -85,B 0,C 180,E1 -26110.983,E2 -26110.983} C_VEL
LIN {X 0,Y 122.59,Z 231.983,A -85,B 0,C 180,E1 -26115.146,E2 -26115.146} C_VEL
LIN {X 0,Y 122.818,Z 233.189,A -85,B 0,C 180,E1 -26116.28,E2 -26116.28} C_VEL
LIN {X 0,Y 125.042,Z 236.74,A -85,B 0,C 180,E1 -26121.428,E2 -26121.428} C_VEL
LIN {X 0,Y 127.406,Z 241.305,A -85,B 0,C 180,E1 -26126.187,E2 -26126.187} C_VEL
LIN {X 0,Y 129.268,Z 245.089,A -85,B 0,C 180,E1 -26129.557,E2 -26129.557} C_VEL
LIN {X 0,Y 131.316,Z 251.271,A -85,B 0,C 180,E1 -26133.869,E2 -26133.869} C_VEL
LIN {X 0,Y 133.066,Z 258.582,A -85,B 0,C 180,E1 -26138.334,E2 -26138.334} C_VEL
LIN {X 0,Y 133.633,Z 264.382,A -85,B 0,C 180,E1 -26141.463,E2 -26141.463} C_VEL
LIN {X 0,Y 133.25,Z 270.427,A -85,B 0,C 180,E1 -26144.394,E2 -26144.394} C_VEL
LIN {X 0,Y 132.18,Z 276.419,A -85,B 0,C 180,E1 -26147.32,E2 -26147.32} C_VEL
LIN {X 0,Y 128.334,Z 283.231,A -85,B 0,C 180,E1 -26150.058,E2 -26150.058} C_VEL
LIN {X 0,Y 123.051,Z 291.305,A -85,B 0,C 180,E1 -26154.168,E2 -26154.168} C_VEL
LIN {X 0,Y 118.857,Z 296.938,A -85,B 0,C 180,E1 -26157.849,E2 -26157.849} C_VEL
LIN {X 0,Y 114.503,Z 302.427,A -85,B 0,C 180,E1 -26162.592,E2 -26162.592} C_VEL
LIN {X 0,Y 110.999,Z 306.729,A -85,B 0,C 180,E1 -26167.674,E2 -26167.674} C_VEL
LIN {X 0,Y 109.143,Z 309.003,A -85,B 0,C 180,E1 -26171.219,E2 -26171.219} C_VEL
LIN {X 0,Y 107.64,Z 310.85,A -85,B 0,C 180,E1 -26174.862,E2 -26174.862} C_VEL
LIN {X 0,Y 106.537,Z 312.234,A -85,B 0,C 180,E1 -26178.587,E2 -26178.587} C_VEL
LIN {X 0,Y 105.777,Z 313.219,A -85,B 0,C 180,E1 -26182.365,E2 -26182.365} C_VEL
LIN {X 0,Y 105.266,Z 314.045,A -85,B 0,C 180,E1 -26190.001,E2 -26190.001} C_VEL
LIN {X 0,Y 105.344,Z 313.849,A -85,B 0,C 180,E1 -26193.826,E2 -26193.826} C_VEL
LIN {X 0,Y 105.777,Z 313.262,A -85,B 0,C 180,E1 -26197.637,E2 -26197.637} C_VEL
LIN {X 0,Y 106.535,Z 312.295,A -85,B 0,C 180,E1 -26201.415,E2 -26201.415} C_VEL
LIN {X 0,Y 107.626,Z 310.938,A -85,B 0,C 180,E1 -26205.142,E2 -26205.142} C_VEL
LIN {X 0,Y 109.964,Z 308.069,A -85,B 0,C 180,E1 -26210.581,E2 -26210.581} C_VEL
LIN {X 0,Y 113.194,Z 304.174,A -85,B 0,C 180,E1 -26215.762,E2 -26215.762} C_VEL
LIN {X 0,Y 117.257,Z 299.147,A -85,B 0,C 180,E1 -26220.629,E2 -26220.629} C_VEL
LIN {X 0,Y 122.102,Z 292.81,A -85,B 0,C 180,E1 -26225.141,E2 -26225.141} C_VEL
LIN {X 0,Y 127.006,Z 285.616,A -85,B 0,C 180,E1 -26229.018,E2 -26229.018} C_VEL
LIN {X 0,Y 132.17,Z 276.817,A -85,B 0,C 180,E1 -26232.686,E2 -26232.686} C_VEL
LIN {X 0,Y 133.447,Z 269.424,A -85,B 0,C 180,E1 -26236.287,E2 -26236.287} C_VEL
LIN {X 0,Y 133.696,Z 263.949,A -85,B 0,C 180,E1 -26238.982,E2 -26238.982} C_VEL
LIN {X 0,Y 133.17,Z 259.003,A -85,B 0,C 180,E1 -26241.676,E2 -26241.676} C_VEL
LIN {X 0,Y 132.038,Z 253.589,A -85,B 0,C 180,E1 -26244.902,E2 -26244.902} C_VEL
LIN {X 0,Y 130.116,Z 247.277,A -85,B 0,C 180,E1 -26249.129,E2 -26249.129} C_VEL
LIN {X 0,Y 129.334,Z 245.111,A -85,B 0,C 180,E1 -26250.721,E2 -26250.721} C_VEL
LIN {X 0,Y 126.801,Z 239.976,A -85,B 0,C 180,E1 -26255.437,E2 -26255.437} C_VEL
LIN {X 0,Y 124.483,Z 235.895,A -85,B 0,C 180,E1 -26260.199,E2 -26260.199} C_VEL
LIN {X 0,Y 123.117,Z 233.852,A -85,B 0,C 180,E1 -26263.416,E2 -26263.416} C_VEL
LIN {X 0,Y 122.202,Z 231.36,A -85,B 0,C 180,E1 -26266.7,E2 -26266.7} C_VEL
LIN {X 0,Y 120.242,Z 228.11,A -85,B 0,C 180,E1 -26280,E2 -26280} C_VEL
LIN {X 0,Y 121.608,Z 231.183,A -85,B 0,C 180,E1 -26290.741,E2 -26290.741} C_VEL
LIN {X 0,Y 122.454,Z 232.209,A -85,B 0,C 180,E1 -26293.272,E2 -26293.272} C_VEL
LIN {X 0,Y 124.028,Z 236.361,A -85,B 0,C 180,E1 -26298.159,E2 -26298.159} C_VEL
LIN {X 0,Y 125.24,Z 238.404,A -85,B 0,C 180,E1 -26300.745,E2 -26300.745} C_VEL
LIN {X 0,Y 126.118,Z 241.091,A -85,B 0,C 180,E1 -26302.959,E2 -26302.959} C_VEL
LIN {X 0,Y 127.347,Z 243.576,A -85,B 0,C 180,E1 -26305.322,E2 -26305.322} C_VEL
LIN {X 0,Y 129.346,Z 249.546,A -85,B 0,C 180,E1 -26309.615,E2 -26309.615} C_VEL
LIN {X 0,Y 131.031,Z 255.289,A -85,B 0,C 180,E1 -26313.286,E2 -26313.286} C_VEL
LIN {X 0,Y 132.566,Z 262.391,A -85,B 0,C 180,E1 -26317.322,E2 -26317.322} C_VEL
LIN {X 0,Y 132.994,Z 266.319,A -85,B 0,C 180,E1 -26319.356,E2 -26319.356} C_VEL
LIN {X 0,Y 132.29,Z 272.396,A -85,B 0,C 180,E1 -26321.947,E2 -26321.947} C_VEL
LIN {X 0,Y 130.368,Z 280.655,A -85,B 0,C 180,E1 -26325.507,E2 -26325.507} C_VEL
LIN {X 0,Y 128.696,Z 285.965,A -85,B 0,C 180,E1 -26328.012,E2 -26328.012} C_VEL
LIN {X 0,Y 127.08,Z 289.19,A -85,B 0,C 180,E1 -26329.471,E2 -26329.471} C_VEL
LIN {X 0,Y 121.546,Z 297.455,A -85,B 0,C 180,E1 -26333.652,E2 -26333.652} C_VEL
LIN {X 0,Y 116.056,Z 305.118,A -85,B 0,C 180,E1 -26339.02,E2 -26339.02} C_VEL
LIN {X 0,Y 112.055,Z 310.221,A -85,B 0,C 180,E1 -26343.957,E2 -26343.957} C_VEL
LIN {X 0,Y 108.898,Z 314.188,A -85,B 0,C 180,E1 -26349.208,E2 -26349.208} C_VEL
LIN {X 0,Y 106.772,Z 317.128,A -85,B 0,C 180,E1 -26354.734,E2 -26354.734} C_VEL
LIN {X 0,Y 105.283,Z 319.53,A -85,B 0,C 180,E1 -26362.327,E2 -26362.327} C_VEL
LIN {X 0,Y 105.046,Z 320.143,A -85,B 0,C 180,E1 -26366.163,E2 -26366.163} C_VEL
LIN {X 0,Y 105.173,Z 320.361,A -85,B 0,C 180,E1 -26369.999,E2 -26369.999} C_VEL
LIN {X 0,Y 105.046,Z 320.129,A -85,B 0,C 180,E1 -26373.835,E2 -26373.835} C_VEL
LIN {X 0,Y 105.283,Z 319.507,A -85,B 0,C 180,E1 -26377.671,E2 -26377.671} C_VEL
LIN {X 0,Y 106.771,Z 317.081,A -85,B 0,C 180,E1 -26385.264,E2 -26385.264} C_VEL
LIN {X 0,Y 108.897,Z 314.121,A -85,B 0,C 180,E1 -26390.79,E2 -26390.79} C_VEL
LIN {X 0,Y 112.052,Z 310.128,A -85,B 0,C 180,E1 -26396.042,E2 -26396.042} C_VEL
LIN {X 0,Y 116.83,Z 303.996,A -85,B 0,C 180,E1 -26401.759,E2 -26401.759} C_VEL
LIN {X 0,Y 121.542,Z 297.297,A -85,B 0,C 180,E1 -26406.347,E2 -26406.347} C_VEL
LIN {X 0,Y 127.052,Z 288.996,A -85,B 0,C 180,E1 -26410.537,E2 -26410.537} C_VEL
LIN {X 0,Y 128.665,Z 285.752,A -85,B 0,C 180,E1 -26411.998,E2 -26411.998} C_VEL
LIN {X 0,Y 131.133,Z 277.359,A -85,B 0,C 180,E1 -26415.835,E2 -26415.835} C_VEL
LIN {X 0,Y 132.59,Z 269.648,A -85,B 0,C 180,E1 -26419.097,E2 -26419.097} C_VEL
LIN {X 0,Y 132.876,Z 264.909,A -85,B 0,C 180,E1 -26421.183,E2 -26421.183} C_VEL
LIN {X 0,Y 131.547,Z 257.826,A -85,B 0,C 180,E1 -26425.11,E2 -26425.11} C_VEL
LIN {X 0,Y 129.865,Z 251.242,A -85,B 0,C 180,E1 -26429.063,E2 -26429.063} C_VEL
LIN {X 0,Y 128.326,Z 246.603,A -85,B 0,C 180,E1 -26432.256,E2 -26432.256} C_VEL
LIN {X 0,Y 126.794,Z 242.441,A -85,B 0,C 180,E1 -26435.436,E2 -26435.436} C_VEL
LIN {X 0,Y 124.577,Z 237.351,A -85,B 0,C 180,E1 -26440.215,E2 -26440.215} C_VEL
LIN {X 0,Y 122.218,Z 232.058,A -85,B 0,C 180,E1 -26446.702,E2 -26446.702} C_VEL
LIN {X 0,Y 120.432,Z 229.624,A -85,B 0,C 180,E1 -26453.298,E2 -26453.298} C_VEL
LIN {X 0,Y 120.055,Z 227.658,A -85,B 0,C 180,E1 -26460,E2 -26460} C_VEL
LIN {X 0,Y 121.914,Z 231.223,A -85,B 0,C 180,E1 -26473.332,E2 -26473.332} C_VEL
LIN {X 0,Y 122.473,Z 232.032,A -85,B 0,C 180,E1 -26474.965,E2 -26474.965} C_VEL
LIN {X 0,Y 122.818,Z 233.189,A -85,B 0,C 180,E1 -26476.28,E2 -26476.28} C_VEL
LIN {X 0,Y 123.542,Z 236.836,A -85,B 0,C 180,E1 -26479.526,E2 -26479.526} C_VEL
LIN {X 0,Y 123.927,Z 241.314,A -85,B 0,C 180,E1 -26482.559,E2 -26482.559} C_VEL
LIN {X 0,Y 124.283,Z 246.031,A -85,B 0,C 180,E1 -26485.545,E2 -26485.545} C_VEL
LIN {X 0,Y 125.022,Z 250.383,A -85,B 0,C 180,E1 -26488.612,E2 -26488.612} C_VEL
LIN {X 0,Y 126.816,Z 257.158,A -85,B 0,C 180,E1 -26493.655,E2 -26493.655} C_VEL
LIN {X 0,Y 127.866,Z 263.387,A -85,B 0,C 180,E1 -26497.735,E2 -26497.735} C_VEL
LIN {X 0,Y 128.015,Z 267.818,A -85,B 0,C 180,E1 -26500.31,E2 -26500.31} C_VEL
LIN {X 0,Y 127.248,Z 273.838,A -85,B 0,C 180,E1 -26503.485,E2 -26503.485} C_VEL
LIN {X 0,Y 126.098,Z 278.404,A -85,B 0,C 180,E1 -26505.84,E2 -26505.84} C_VEL
LIN {X 0,Y 120.838,Z 286.651,A -85,B 0,C 180,E1 -26509.442,E2 -26509.442} C_VEL
LIN {X 0,Y 115.52,Z 293.91,A -85,B 0,C 180,E1 -26513.619,E2 -26513.619} C_VEL
LIN {X 0,Y 109.664,Z 300.956,A -85,B 0,C 180,E1 -26519.158,E2 -26519.158} C_VEL
LIN {X 0,Y 105.649,Z 305.638,A -85,B 0,C 180,E1 -26524.382,E2 -26524.382} C_VEL
LIN {X 0,Y 102.451,Z 309.217,A -85,B 0,C 180,E1 -26529.942,E2 -26529.942} C_VEL
LIN {X 0,Y 100.806,Z 311.064,A -85,B 0,C 180,E1 -26533.808,E2 -26533.808} C_VEL
LIN {X 0,Y 99.579,Z 312.448,A -85,B 0,C 180,E1 -26537.777,E2 -26537.777} C_VEL
LIN {X 0,Y 98.755,Z 313.432,A -85,B 0,C 180,E1 -26541.818,E2 -26541.818} C_VEL
LIN {X 0,Y 98.192,Z 314.257,A -85,B 0,C 180,E1 -26550.001,E2 -26550.001} C_VEL
LIN {X 0,Y 98.755,Z 313.475,A -85,B 0,C 180,E1 -26558.184,E2 -26558.184} C_VEL
LIN {X 0,Y 100.793,Z 311.15,A -85,B 0,C 180,E1 -26566.196,E2 -26566.196} C_VEL
LIN {X 0,Y 103.343,Z 308.281,A -85,B 0,C 180,E1 -26571.966,E2 -26571.966} C_VEL
LIN {X 0,Y 106.825,Z 304.387,A -85,B 0,C 180,E1 -26577.422,E2 -26577.422} C_VEL
LIN {X 0,Y 111.213,Z 299.359,A -85,B 0,C 180,E1 -26582.491,E2 -26582.491} C_VEL
LIN {X 0,Y 116.368,Z 293.021,A -85,B 0,C 180,E1 -26587.154,E2 -26587.154} C_VEL
LIN {X 0,Y 122.463,Z 284.491,A -85,B 0,C 180,E1 -26591.75,E2 -26591.75} C_VEL
LIN {X 0,Y 126.072,Z 278.797,A -85,B 0,C 180,E1 -26594.174,E2 -26594.174} C_VEL
LIN {X 0,Y 127.249,Z 274.233,A -85,B 0,C 180,E1 -26596.536,E2 -26596.536} C_VEL
LIN {X 0,Y 128.103,Z 268.204,A -85,B 0,C 180,E1 -26599.69,E2 -26599.69} C_VEL
LIN {X 0,Y 127.869,Z 262.949,A -85,B 0,C 180,E1 -26602.8,E2 -26602.8} C_VEL
LIN {X 0,Y 126.674,Z 256.223,A -85,B 0,C 180,E1 -26607.252,E2 -26607.252} C_VEL
LIN {X 0,Y 125.159,Z 250.631,A -85,B 0,C 180,E1 -26611.491,E2 -26611.491} C_VEL
LIN {X 0,Y 123.307,Z 246.207,A -85,B 0,C 180,E1 -26615.776,E2 -26615.776} C_VEL
LIN {X 0,Y 121.725,Z 242.857,A -85,B 0,C 180,E1 -26619.731,E2 -26619.731} C_VEL
LIN {X 0,Y 119.676,Z 238.346,A -85,B 0,C 180,E1 -26626.414,E2 -26626.414} C_VEL
LIN {X 0,Y 118.064,Z 236.447,A -85,B 0,C 180,E1 -26633.162,E2 -26633.162} C_VEL
LIN {X 0,Y 117.988,Z 234.889,A -85,B 0,C 180,E1 -26640,E2 -26640} C_VEL
LIN {X 0,Y 119.019,Z 237.688,A -85,B 0,C 180,E1 -26650.204,E2 -26650.204} C_VEL
LIN {X 0,Y 119.91,Z 239.355,A -85,B 0,C 180,E1 -26653.559,E2 -26653.559} C_VEL
LIN {X 0,Y 121.936,Z 244.798,A -85,B 0,C 180,E1 -26660.232,E2 -26660.232} C_VEL
LIN {X 0,Y 123.444,Z 249.167,A -85,B 0,C 180,E1 -26664.365,E2 -26664.365} C_VEL
LIN {X 0,Y 125.332,Z 255.94,A -85,B 0,C 180,E1 -26669.57,E2 -26669.57} C_VEL
LIN {X 0,Y 126.619,Z 262.244,A -85,B 0,C 180,E1 -26673.714,E2 -26673.714} C_VEL
LIN {X 0,Y 127.391,Z 268.304,A -85,B 0,C 180,E1 -26677.363,E2 -26677.363} C_VEL
LIN {X 0,Y 127.079,Z 272.16,A -85,B 0,C 180,E1 -26679.261,E2 -26679.261} C_VEL
LIN {X 0,Y 125.02,Z 280.429,A -85,B 0,C 180,E1 -26683.046,E2 -26683.046} C_VEL
LIN {X 0,Y 122.564,Z 287.392,A -85,B 0,C 180,E1 -26686.519,E2 -26686.519} C_VEL
LIN {X 0,Y 119.694,Z 291.957,A -85,B 0,C 180,E1 -26688.657,E2 -26688.657} C_VEL
LIN {X 0,Y 114.99,Z 298.481,A -85,B 0,C 180,E1 -26692.324,E2 -26692.324} C_VEL
LIN {X 0,Y 110.03,Z 304.906,A -85,B 0,C 180,E1 -26697.116,E2 -26697.116} C_VEL
LIN {X 0,Y 105.704,Z 310.008,A -85,B 0,C 180,E1 -26702.262,E2 -26702.262} C_VEL
LIN {X 0,Y 102.266,Z 313.975,A -85,B 0,C 180,E1 -26707.791,E2 -26707.791} C_VEL
LIN {X 0,Y 99.898,Z 316.914,A -85,B 0,C 180,E1 -26713.655,E2 -26713.655} C_VEL
LIN {X 0,Y 98.871,Z 318.314,A -85,B 0,C 180,E1 -26717.686,E2 -26717.686} C_VEL
LIN {X 0,Y 98.251,Z 319.318,A -85,B 0,C 180,E1 -26721.774,E2 -26721.774} C_VEL
LIN {X 0,Y 97.952,Z 319.93,A -85,B 0,C 180,E1 -26725.885,E2 -26725.885} C_VEL
LIN {X 0,Y 98.077,Z 320.148,A -85,B 0,C 180,E1 -26729.999,E2 -26729.999} C_VEL
LIN {X 0,Y 98.25,Z 319.293,A -85,B 0,C 180,E1 -26738.224,E2 -26738.224} C_VEL
LIN {X 0,Y 98.87,Z 318.281,A -85,B 0,C 180,E1 -26742.312,E2 -26742.312} C_VEL
LIN {X 0,Y 99.897,Z 316.865,A -85,B 0,C 180,E1 -26746.343,E2 -26746.343} C_VEL
LIN {X 0,Y 102.265,Z 313.906,A -85,B 0,C 180,E1 -26752.207,E2 -26752.207} C_VEL
LIN {X 0,Y 105.701,Z 309.913,A -85,B 0,C 180,E1 -26757.737,E2 -26757.737} C_VEL
LIN {X 0,Y 110.821,Z 303.779,A -85,B 0,C 180,E1 -26763.703,E2 -26763.703} C_VEL
LIN {X 0,Y 115.852,Z 297.08,A -85,B 0,C 180,E1 -26768.447,E2 -26768.447} C_VEL
LIN {X 0,Y 121.691,Z 288.778,A -85,B 0,C 180,E1 -26772.733,E2 -26772.733} C_VEL
LIN {X 0,Y 123.811,Z 283.814,A -85,B 0,C 180,E1 -26775.197,E2 -26775.197} C_VEL
LIN {X 0,Y 126.313,Z 275.121,A -85,B 0,C 180,E1 -26779.3,E2 -26779.3} C_VEL
LIN {X 0,Y 127.363,Z 269.099,A -85,B 0,C 180,E1 -26782.05,E2 -26782.05} C_VEL
LIN {X 0,Y 126.733,Z 263.479,A -85,B 0,C 180,E1 -26785.36,E2 -26785.36} C_VEL
LIN {X 0,Y 125.451,Z 256.719,A -85,B 0,C 180,E1 -26789.722,E2 -26789.722} C_VEL
LIN {X 0,Y 123.539,Z 249.781,A -85,B 0,C 180,E1 -26794.924,E2 -26794.924} C_VEL
LIN {X 0,Y 121.752,Z 244.609,A -85,B 0,C 180,E1 -26799.736,E2 -26799.736} C_VEL
LIN {X 0,Y 119.722,Z 239.095,A -85,B 0,C 180,E1 -26806.42,E2 -26806.42} C_VEL
LIN {X 0,Y 118.795,Z 237.504,A -85,B 0,C 180,E1 -26809.777,E2 -26809.777} C_VEL
LIN {X 0,Y 117.83,Z 234.453,A -85,B 0,C 180,E1 -26820,E2 -26820} C_VEL
LIN {X 0,Y 119.453,Z 238.058,A -85,B 0,C 180,E1 -26833.612,E2 -26833.612} C_VEL
LIN {X 0,Y 121.535,Z 242.52,A -85,B 0,C 180,E1 -26840.302,E2 -26840.302} C_VEL
LIN {X 0,Y 123.525,Z 246.898,A -85,B 0,C 180,E1 -26845.258,E2 -26845.258} C_VEL
LIN {X 0,Y 125.022,Z 250.383,A -85,B 0,C 180,E1 -26848.612,E2 -26848.612} C_VEL
LIN {X 0,Y 125.485,Z 253.776,A -85,B 0,C 180,E1 -26850.825,E2 -26850.825} C_VEL
LIN {X 0,Y 125.018,Z 259.171,A -85,B 0,C 180,E1 -26853.487,E2 -26853.487} C_VEL
LIN {X 0,Y 123.46,Z 266.387,A -85,B 0,C 180,E1 -26856.69,E2 -26856.69} C_VEL
LIN {X 0,Y 122.27,Z 271.82,A -85,B 0,C 180,E1 -26859.452,E2 -26859.452} C_VEL
LIN {X 0,Y 120.78,Z 278.635,A -85,B 0,C 180,E1 -26863.336,E2 -26863.336} C_VEL
LIN {X 0,Y 120.053,Z 280.3,A -85,B 0,C 180,E1 -26864.184,E2 -26864.184} C_VEL
LIN {X 0,Y 113.772,Z 289.19,A -85,B 0,C 180,E1 -26868.391,E2 -26868.391} C_VEL
LIN {X 0,Y 108.015,Z 296.345,A -85,B 0,C 180,E1 -26872.999,E2 -26872.999} C_VEL
LIN {X 0,Y 103.636,Z 301.17,A -85,B 0,C 180,E1 -26877.146,E2 -26877.146} C_VEL
LIN {X 0,Y 99.297,Z 305.852,A -85,B 0,C 180,E1 -26882.611,E2 -26882.611} C_VEL
LIN {X 0,Y 95.793,Z 309.432,A -85,B 0,C 180,E1 -26888.481,E2 -26888.481} C_VEL
LIN {X 0,Y 93.998,Z 311.278,A -85,B 0,C 180,E1 -26892.599,E2 -26892.599} C_VEL
LIN {X 0,Y 92.658,Z 312.661,A -85,B 0,C 180,E1 -26896.849,E2 -26896.849} C_VEL
LIN {X 0,Y 91.732,Z 313.645,A -85,B 0,C 180,E1 -26901.187,E2 -26901.187} C_VEL
LIN {X 0,Y 91.114,Z 314.47,A -85,B 0,C 180,E1 -26910.001,E2 -26910.001} C_VEL
LIN {X 0,Y 91.207,Z 314.274,A -85,B 0,C 180,E1 -26914.42,E2 -26914.42} C_VEL
LIN {X 0,Y 91.732,Z 313.687,A -85,B 0,C 180,E1 -26918.815,E2 -26918.815} C_VEL
LIN {X 0,Y 92.656,Z 312.72,A -85,B 0,C 180,E1 -26923.154,E2 -26923.154} C_VEL
LIN {X 0,Y 93.982,Z 311.363,A -85,B 0,C 180,E1 -26927.406,E2 -26927.406} C_VEL
LIN {X 0,Y 96.798,Z 308.493,A -85,B 0,C 180,E1 -26933.537,E2 -26933.537} C_VEL
LIN {X 0,Y 100.559,Z 304.599,A -85,B 0,C 180,E1 -26939.291,E2 -26939.291} C_VEL
LIN {X 0,Y 105.302,Z 299.57,A -85,B 0,C 180,E1 -26944.563,E2 -26944.563} C_VEL
LIN {X 0,Y 110.79,Z 293.232,A -85,B 0,C 180,E1 -26949.373,E2 -26949.373} C_VEL
LIN {X 0,Y 116.943,Z 285.15,A -85,B 0,C 180,E1 -26953.848,E2 -26953.848} C_VEL
LIN {X 0,Y 120.004,Z 280.655,A -85,B 0,C 180,E1 -26955.842,E2 -26955.842} C_VEL
LIN {X 0,Y 120.805,Z 279.019,A -85,B 0,C 180,E1 -26956.654,E2 -26956.654} C_VEL
LIN {X 0,Y 122.287,Z 272.519,A -85,B 0,C 180,E1 -26960.349,E2 -26960.349} C_VEL
LIN {X 0,Y 122.541,Z 267.633,A -85,B 0,C 180,E1 -26963.412,E2 -26963.412} C_VEL
LIN {X 0,Y 121.902,Z 261.509,A -85,B 0,C 180,E1 -26967.772,E2 -26967.772} C_VEL
LIN {X 0,Y 120.789,Z 255.991,A -85,B 0,C 180,E1 -26972.259,E2 -26972.259} C_VEL
LIN {X 0,Y 119.664,Z 252.557,A -85,B 0,C 180,E1 -26975.725,E2 -26975.725} C_VEL
LIN {X 0,Y 117.984,Z 248.518,A -85,B 0,C 180,E1 -26980.875,E2 -26980.875} C_VEL
LIN {X 0,Y 116.655,Z 245.319,A -85,B 0,C 180,E1 -26986.055,E2 -26986.055} C_VEL
LIN {X 0,Y 115.942,Z 243.873,A -85,B 0,C 180,E1 -26989.522,E2 -26989.522} C_VEL
LIN {X 0,Y 115.321,Z 241.519,A -85,B 0,C 180,E1 -27000,E2 -27000} C_VEL
LIN {X 0,Y 116.237,Z 244.42,A -85,B 0,C 180,E1 -27010.451,E2 -27010.451} C_VEL
LIN {X 0,Y 116.609,Z 245.254,A -85,B 0,C 180,E1 -27012.178,E2 -27012.178} C_VEL
LIN {X 0,Y 118.178,Z 250.359,A -85,B 0,C 180,E1 -27019.092,E2 -27019.092} C_VEL
LIN {X 0,Y 119.099,Z 253.701,A -85,B 0,C 180,E1 -27022.554,E2 -27022.554} C_VEL
LIN {X 0,Y 120.239,Z 258.767,A -85,B 0,C 180,E1 -27026.936,E2 -27026.936} C_VEL
LIN {X 0,Y 121.261,Z 264.784,A -85,B 0,C 180,E1 -27031.441,E2 -27031.441} C_VEL
LIN {X 0,Y 121.823,Z 270.429,A -85,B 0,C 180,E1 -27035.233,E2 -27035.233} C_VEL
LIN {X 0,Y 121.692,Z 273.619,A -85,B 0,C 180,E1 -27037.127,E2 -27037.127} C_VEL
LIN {X 0,Y 119.528,Z 281.231,A -85,B 0,C 180,E1 -27040.881,E2 -27040.881} C_VEL
LIN {X 0,Y 116.484,Z 288.762,A -85,B 0,C 180,E1 -27044.851,E2 -27044.851} C_VEL
LIN {X 0,Y 111.348,Z 295.793,A -85,B 0,C 180,E1 -27048.491,E2 -27048.491} C_VEL
LIN {X 0,Y 105.797,Z 302.685,A -85,B 0,C 180,E1 -27053.282,E2 -27053.282} C_VEL
LIN {X 0,Y 100.852,Z 308.205,A -85,B 0,C 180,E1 -27058.489,E2 -27058.489} C_VEL
LIN {X 0,Y 96.837,Z 312.539,A -85,B 0,C 180,E1 -27064.185,E2 -27064.185} C_VEL
LIN {X 0,Y 94.688,Z 314.837,A -85,B 0,C 180,E1 -27068.215,E2 -27068.215} C_VEL
LIN {X 0,Y 93.07,Z 316.7,A -85,B 0,C 180,E1 -27072.418,E2 -27072.418} C_VEL
LIN {X 0,Y 91.219,Z 319.104,A -85,B 0,C 180,E1 -27081.135,E2 -27081.135} C_VEL
LIN {X 0,Y 90.882,Z 319.717,A -85,B 0,C 180,E1 -27085.564,E2 -27085.564} C_VEL
LIN {X 0,Y 90.975,Z 319.935,A -85,B 0,C 180,E1 -27089.999,E2 -27089.999} C_VEL
LIN {X 0,Y 90.881,Z 319.702,A -85,B 0,C 180,E1 -27094.434,E2 -27094.434} C_VEL
LIN {X 0,Y 91.218,Z 319.08,A -85,B 0,C 180,E1 -27098.863,E2 -27098.863} C_VEL
LIN {X 0,Y 91.914,Z 318.067,A -85,B 0,C 180,E1 -27103.26,E2 -27103.26} C_VEL
LIN {X 0,Y 93.069,Z 316.65,A -85,B 0,C 180,E1 -27107.58,E2 -27107.58} C_VEL
LIN {X 0,Y 95.712,Z 313.691,A -85,B 0,C 180,E1 -27113.818,E2 -27113.818} C_VEL
LIN {X 0,Y 99.437,Z 309.698,A -85,B 0,C 180,E1 -27119.652,E2 -27119.652} C_VEL
LIN {X 0,Y 104.961,Z 303.564,A -85,B 0,C 180,E1 -27125.864,E2 -27125.864} C_VEL
LIN {X 0,Y 110.344,Z 296.863,A -85,B 0,C 180,E1 -27130.755,E2 -27130.755} C_VEL
LIN {X 0,Y 116.463,Z 288.558,A -85,B 0,C 180,E1 -27135.157,E2 -27135.157} C_VEL
LIN {X 0,Y 119.423,Z 281.123,A -85,B 0,C 180,E1 -27139.075,E2 -27139.075} C_VEL
LIN {X 0,Y 121.513,Z 273.798,A -85,B 0,C 180,E1 -27142.677,E2 -27142.677} C_VEL
LIN {X 0,Y 121.817,Z 271.6,A -85,B 0,C 180,E1 -27143.871,E2 -27143.871} C_VEL
LIN {X 0,Y 121.12,Z 264.645,A -85,B 0,C 180,E1 -27148.518,E2 -27148.518} C_VEL
LIN {X 0,Y 120.333,Z 259.695,A -85,B 0,C 180,E1 -27152.145,E2 -27152.145} C_VEL
LIN {X 0,Y 119.433,Z 255.403,A -85,B 0,C 180,E1 -27155.675,E2 -27155.675} C_VEL
LIN {X 0,Y 117.997,Z 250.18,A -85,B 0,C 180,E1 -27160.878,E2 -27160.878} C_VEL
LIN {X 0,Y 116.746,Z 246.183,A -85,B 0,C 180,E1 -27166.067,E2 -27166.067} C_VEL
LIN {X 0,Y 116.024,Z 244.236,A -85,B 0,C 180,E1 -27169.53,E2 -27169.53} C_VEL
LIN {X 0,Y 115.188,Z 241.102,A -85,B 0,C 180,E1 -27180,E2 -27180} C_VEL
LIN {X 0,Y 115.709,Z 243.655,A -85,B 0,C 180,E1 -27190.499,E2 -27190.499} C_VEL
LIN {X 0,Y 116.486,Z 244.989,A -85,B 0,C 180,E1 -27193.966,E2 -27193.966} C_VEL
LIN {X 0,Y 117.797,Z 248.219,A -85,B 0,C 180,E1 -27199.156,E2 -27199.156} C_VEL
LIN {X 0,Y 119.448,Z 252.346,A -85,B 0,C 180,E1 -27204.322,E2 -27204.322} C_VEL
LIN {X 0,Y 120.855,Z 256.69,A -85,B 0,C 180,E1 -27208.626,E2 -27208.626} C_VEL
LIN {X 0,Y 121.845,Z 261.741,A -85,B 0,C 180,E1 -27212.661,E2 -27212.661} C_VEL
LIN {X 0,Y 122.457,Z 267.179,A -85,B 0,C 180,E1 -27216.538,E2 -27216.538} C_VEL
LIN {X 0,Y 122.27,Z 271.82,A -85,B 0,C 180,E1 -27219.452,E2 -27219.452} C_VEL
LIN {X 0,Y 121.431,Z 274.493,A -85,B 0,C 180,E1 -27220.772,E2 -27220.772} C_VEL
LIN {X 0,Y 118.984,Z 278.697,A -85,B 0,C 180,E1 -27222.399,E2 -27222.399} C_VEL
LIN {X 0,Y 115.621,Z 282.828,A -85,B 0,C 180,E1 -27223.778,E2 -27223.778} C_VEL
LIN {X 0,Y 107.896,Z 290.608,A -85,B 0,C 180,E1 -27226.74,E2 -27226.74} C_VEL
LIN {X 0,Y 105.635,Z 292.95,A -85,B 0,C 180,E1 -27228.057,E2 -27228.057} C_VEL
LIN {X 0,Y 99.586,Z 299.578,A -85,B 0,C 180,E1 -27233.141,E2 -27233.141} C_VEL
LIN {X 0,Y 94.486,Z 304.654,A -85,B 0,C 180,E1 -27238.624,E2 -27238.624} C_VEL
LIN {X 0,Y 90.378,Z 308.589,A -85,B 0,C 180,E1 -27244.68,E2 -27244.68} C_VEL
LIN {X 0,Y 87.246,Z 311.492,A -85,B 0,C 180,E1 -27251.204,E2 -27251.204} C_VEL
LIN {X 0,Y 85.755,Z 312.875,A -85,B 0,C 180,E1 -27255.768,E2 -27255.768} C_VEL
LIN {X 0,Y 84.74,Z 313.858,A -85,B 0,C 180,E1 -27260.453,E2 -27260.453} C_VEL
LIN {X 0,Y 84.024,Z 314.682,A -85,B 0,C 180,E1 -27270.001,E2 -27270.001} C_VEL
LIN {X 0,Y 84.74,Z 313.9,A -85,B 0,C 180,E1 -27279.549,E2 -27279.549} C_VEL
LIN {X 0,Y 87.23,Z 311.575,A -85,B 0,C 180,E1 -27288.802,E2 -27288.802} C_VEL
LIN {X 0,Y 90.342,Z 308.705,A -85,B 0,C 180,E1 -27295.333,E2 -27295.333} C_VEL
LIN {X 0,Y 94.417,Z 304.812,A -85,B 0,C 180,E1 -27301.404,E2 -27301.404} C_VEL
LIN {X 0,Y 99.547,Z 299.781,A -85,B 0,C 180,E1 -27306.878,E2 -27306.878} C_VEL
LIN {X 0,Y 105.397,Z 293.443,A -85,B 0,C 180,E1 -27311.822,E2 -27311.822} C_VEL
LIN {X 0,Y 111.57,Z 285.839,A -85,B 0,C 180,E1 -27316.138,E2 -27316.138} C_VEL
LIN {X 0,Y 115.021,Z 280.872,A -85,B 0,C 180,E1 -27318.462,E2 -27318.462} C_VEL
LIN {X 0,Y 116.764,Z 274.601,A -85,B 0,C 180,E1 -27322.357,E2 -27322.357} C_VEL
LIN {X 0,Y 117.073,Z 270.522,A -85,B 0,C 180,E1 -27325.231,E2 -27325.231} C_VEL
LIN {X 0,Y 116.81,Z 265.646,A -85,B 0,C 180,E1 -27329.085,E2 -27329.085} C_VEL
LIN {X 0,Y 116.214,Z 261.207,A -85,B 0,C 180,E1 -27333.027,E2 -27333.027} C_VEL
LIN {X 0,Y 115.416,Z 258.021,A -85,B 0,C 180,E1 -27336.494,E2 -27336.494} C_VEL
LIN {X 0,Y 114.027,Z 254.047,A -85,B 0,C 180,E1 -27342.051,E2 -27342.051} C_VEL
LIN {X 0,Y 113.273,Z 252.012,A -85,B 0,C 180,E1 -27345.63,E2 -27345.63} C_VEL
LIN {X 0,Y 112.743,Z 250.373,A -85,B 0,C 180,E1 -27349.221,E2 -27349.221} C_VEL
LIN {X 0,Y 112.288,Z 248.006,A -85,B 0,C 180,E1 -27360,E2 -27360} C_VEL
LIN {X 0,Y 112.503,Z 249.754,A -85,B 0,C 180,E1 -27367.177,E2 -27367.177} C_VEL
LIN {X 0,Y 113.077,Z 250.989,A -85,B 0,C 180,E1 -27370.746,E2 -27370.746} C_VEL
LIN {X 0,Y 114.202,Z 255.782,A -85,B 0,C 180,E1 -27377.921,E2 -27377.921} C_VEL
LIN {X 0,Y 115.041,Z 260.175,A -85,B 0,C 180,E1 -27382.68,E2 -27382.68} C_VEL
LIN {X 0,Y 115.742,Z 265.083,A -85,B 0,C 180,E1 -27387.091,E2 -27387.091} C_VEL
LIN {X 0,Y 116.276,Z 271.615,A -85,B 0,C 180,E1 -27392.199,E2 -27392.199} C_VEL
LIN {X 0,Y 116.266,Z 275.434,A -85,B 0,C 180,E1 -27394.896,E2 -27394.896} C_VEL
LIN {X 0,Y 114.962,Z 279.969,A -85,B 0,C 180,E1 -27397.369,E2 -27397.369} C_VEL
LIN {X 0,Y 112.097,Z 286.945,A -85,B 0,C 180,E1 -27401.205,E2 -27401.205} C_VEL
LIN {X 0,Y 110.477,Z 290.044,A -85,B 0,C 180,E1 -27402.981,E2 -27402.981} C_VEL
LIN {X 0,Y 104.038,Z 298.056,A -85,B 0,C 180,E1 -27407.504,E2 -27407.504} C_VEL
LIN {X 0,Y 98.38,Z 304.482,A -85,B 0,C 180,E1 -27412.611,E2 -27412.611} C_VEL
LIN {X 0,Y 93.292,Z 309.582,A -85,B 0,C 180,E1 -27418.174,E2 -27418.174} C_VEL
LIN {X 0,Y 89.227,Z 313.549,A -85,B 0,C 180,E1 -27424.327,E2 -27424.327} C_VEL
LIN {X 0,Y 86.3,Z 316.487,A -85,B 0,C 180,E1 -27430.988,E2 -27430.988} C_VEL
LIN {X 0,Y 84.192,Z 318.891,A -85,B 0,C 180,E1 -27440.388,E2 -27440.388} C_VEL
LIN {X 0,Y 83.799,Z 319.504,A -85,B 0,C 180,E1 -27445.188,E2 -27445.188} C_VEL
LIN {X 0,Y 83.881,Z 319.722,A -85,B 0,C 180,E1 -27449.999,E2 -27449.999} C_VEL
LIN {X 0,Y 83.799,Z 319.489,A -85,B 0,C 180,E1 -27454.81,E2 -27454.81} C_VEL
LIN {X 0,Y 84.192,Z 318.866,A -85,B 0,C 180,E1 -27459.609,E2 -27459.609} C_VEL
LIN {X 0,Y 84.999,Z 317.852,A -85,B 0,C 180,E1 -27464.361,E2 -27464.361} C_VEL
LIN {X 0,Y 86.299,Z 316.436,A -85,B 0,C 180,E1 -27469.01,E2 -27469.01} C_VEL
LIN {X 0,Y 89.225,Z 313.476,A -85,B 0,C 180,E1 -27475.671,E2 -27475.671} C_VEL
LIN {X 0,Y 93.289,Z 309.482,A -85,B 0,C 180,E1 -27481.825,E2 -27481.825} C_VEL
LIN {X 0,Y 99.272,Z 303.348,A -85,B 0,C 180,E1 -27488.275,E2 -27488.275} C_VEL
LIN {X 0,Y 105.037,Z 296.647,A -85,B 0,C 180,E1 -27493.299,E2 -27493.299} C_VEL
LIN {X 0,Y 110.455,Z 289.835,A -85,B 0,C 180,E1 -27497.029,E2 -27497.029} C_VEL
LIN {X 0,Y 113.303,Z 283.924,A -85,B 0,C 180,E1 -27500.386,E2 -27500.386} C_VEL
LIN {X 0,Y 115.901,Z 276.573,A -85,B 0,C 180,E1 -27504.301,E2 -27504.301} C_VEL
LIN {X 0,Y 116.245,Z 275.118,A -85,B 0,C 180,E1 -27505.123,E2 -27505.123} C_VEL
LIN {X 0,Y 116.009,Z 269.047,A -85,B 0,C 180,E1 -27509.565,E2 -27509.565} C_VEL
LIN {X 0,Y 115.496,Z 263.744,A -85,B 0,C 180,E1 -27513.822,E2 -27513.822} C_VEL
LIN {X 0,Y 114.708,Z 258.799,A -85,B 0,C 180,E1 -27518.432,E2 -27518.432} C_VEL
LIN {X 0,Y 114.023,Z 255.615,A -85,B 0,C 180,E1 -27522.05,E2 -27522.05} C_VEL
LIN {X 0,Y 113.111,Z 251.814,A -85,B 0,C 180,E1 -27527.44,E2 -27527.44} C_VEL
LIN {X 0,Y 112.848,Z 250.874,A -85,B 0,C 180,E1 -27529.232,E2 -27529.232} C_VEL
LIN {X 0,Y 112.32,Z 249.519,A -85,B 0,C 180,E1 -27532.811,E2 -27532.811} C_VEL
LIN {X 0,Y 112.177,Z 247.598,A -85,B 0,C 180,E1 -27540,E2 -27540} C_VEL
LIN {X 0,Y 112.547,Z 250.137,A -85,B 0,C 180,E1 -27550.798,E2 -27550.798} C_VEL
LIN {X 0,Y 113.369,Z 252.712,A -85,B 0,C 180,E1 -27556.053,E2 -27556.053} C_VEL
LIN {X 0,Y 114.231,Z 254.995,A -85,B 0,C 180,E1 -27559.779,E2 -27559.779} C_VEL
LIN {X 0,Y 115.585,Z 259.289,A -85,B 0,C 180,E1 -27565.191,E2 -27565.191} C_VEL
LIN {X 0,Y 116.218,Z 261.961,A -85,B 0,C 180,E1 -27567.948,E2 -27567.948} C_VEL
LIN {X 0,Y 116.866,Z 267.624,A -85,B 0,C 180,E1 -27572.768,E2 -27572.768} C_VEL
LIN {X 0,Y 116.969,Z 271.672,A -85,B 0,C 180,E1 -27575.862,E2 -27575.862} C_VEL
LIN {X 0,Y 116.475,Z 275.373,A -85,B 0,C 180,E1 -27578.336,E2 -27578.336} C_VEL
LIN {X 0,Y 115.01,Z 280.526,A -85,B 0,C 180,E1 -27581.535,E2 -27581.535} C_VEL
LIN {X 0,Y 112.223,Z 284.656,A -85,B 0,C 180,E1 -27583.452,E2 -27583.452} C_VEL
LIN {X 0,Y 105.635,Z 292.95,A -85,B 0,C 180,E1 -27588.057,E2 -27588.057} C_VEL
LIN {X 0,Y 102.208,Z 296.207,A -85,B 0,C 180,E1 -27590.02,E2 -27590.02} C_VEL
LIN {X 0,Y 95.354,Z 301.007,A -85,B 0,C 180,E1 -27593.117,E2 -27593.117} C_VEL
LIN {X 0,Y 88.71,Z 305.154,A -85,B 0,C 180,E1 -27596.908,E2 -27596.908} C_VEL
LIN {X 0,Y 85.747,Z 307.295,A -85,B 0,C 180,E1 -27599.943,E2 -27599.943} C_VEL
LIN {X 0,Y 82.742,Z 309.86,A -85,B 0,C 180,E1 -27604.87,E2 -27604.87} C_VEL
LIN {X 0,Y 80.564,Z 311.705,A -85,B 0,C 180,E1 -27609.579,E2 -27609.579} C_VEL
LIN {X 0,Y 77.747,Z 314.072,A -85,B 0,C 180,E1 -27619.586,E2 -27619.586} C_VEL
LIN {X 0,Y 76.925,Z 314.896,A -85,B 0,C 180,E1 -27630.001,E2 -27630.001} C_VEL
LIN {X 0,Y 77.072,Z 314.699,A -85,B 0,C 180,E1 -27635.233,E2 -27635.233} C_VEL
LIN {X 0,Y 77.747,Z 314.112,A -85,B 0,C 180,E1 -27640.417,E2 -27640.417} C_VEL
LIN {X 0,Y 80.548,Z 311.787,A -85,B 0,C 180,E1 -27650.428,E2 -27650.428} C_VEL
LIN {X 0,Y 83.973,Z 308.918,A -85,B 0,C 180,E1 -27657.409,E2 -27657.409} C_VEL
LIN {X 0,Y 88.423,Z 305.024,A -85,B 0,C 180,E1 -27663.806,E2 -27663.806} C_VEL
LIN {X 0,Y 93.974,Z 299.992,A -85,B 0,C 180,E1 -27669.472,E2 -27669.472} C_VEL
LIN {X 0,Y 100.216,Z 293.654,A -85,B 0,C 180,E1 -27674.531,E2 -27674.531} C_VEL
LIN {X 0,Y 106.372,Z 286.552,A -85,B 0,C 180,E1 -27678.646,E2 -27678.646} C_VEL
LIN {X 0,Y 109.321,Z 282.698,A -85,B 0,C 180,E1 -27680.486,E2 -27680.486} C_VEL
LIN {X 0,Y 111.084,Z 277.706,A -85,B 0,C 180,E1 -27683.81,E2 -27683.81} C_VEL
LIN {X 0,Y 111.618,Z 273.581,A -85,B 0,C 180,E1 -27687.045,E2 -27687.045} C_VEL
LIN {X 0,Y 111.612,Z 269.333,A -85,B 0,C 180,E1 -27690.82,E2 -27690.82} C_VEL
LIN {X 0,Y 111.44,Z 266.26,A -85,B 0,C 180,E1 -27693.803,E2 -27693.803} C_VEL
LIN {X 0,Y 110.858,Z 263.054,A -85,B 0,C 180,E1 -27697.643,E2 -27697.643} C_VEL
LIN {X 0,Y 109.761,Z 259.133,A -85,B 0,C 180,E1 -27703.835,E2 -27703.835} C_VEL
LIN {X 0,Y 109.142,Z 256.729,A -85,B 0,C 180,E1 -27708.861,E2 -27708.861} C_VEL
LIN {X 0,Y 108.624,Z 255.006,A -85,B 0,C 180,E1 -27716.29,E2 -27716.29} C_VEL
LIN {X 0,Y 108.911,Z 254.305,A -85,B 0,C 180,E1 -27720,E2 -27720} C_VEL
LIN {X 0,Y 109.036,Z 256.07,A -85,B 0,C 180,E1 -27727.407,E2 -27727.407} C_VEL
LIN {X 0,Y 109.432,Z 257.485,A -85,B 0,C 180,E1 -27731.108,E2 -27731.108} C_VEL
LIN {X 0,Y 109.983,Z 260.951,A -85,B 0,C 180,E1 -27736.56,E2 -27736.56} C_VEL
LIN {X 0,Y 110.395,Z 264.135,A -85,B 0,C 180,E1 -27740.496,E2 -27740.496} C_VEL
LIN {X 0,Y 110.735,Z 268.435,A -85,B 0,C 180,E1 -27744.858,E2 -27744.858} C_VEL
LIN {X 0,Y 110.891,Z 273.583,A -85,B 0,C 180,E1 -27749.417,E2 -27749.417} C_VEL
LIN {X 0,Y 110.679,Z 278.336,A -85,B 0,C 180,E1 -27753.208,E2 -27753.208} C_VEL
LIN {X 0,Y 109.443,Z 281.861,A -85,B 0,C 180,E1 -27755.306,E2 -27755.306} C_VEL
LIN {X 0,Y 105.589,Z 289.826,A -85,B 0,C 180,E1 -27760.053,E2 -27760.053} C_VEL
LIN {X 0,Y 103.419,Z 292.695,A -85,B 0,C 180,E1 -27761.622,E2 -27761.622} C_VEL
LIN {X 0,Y 96.552,Z 300.346,A -85,B 0,C 180,E1 -27766.537,E2 -27766.537} C_VEL
LIN {X 0,Y 90.875,Z 306.09,A -85,B 0,C 180,E1 -27771.778,E2 -27771.778} C_VEL
LIN {X 0,Y 85.723,Z 310.804,A -85,B 0,C 180,E1 -27777.797,E2 -27777.797} C_VEL
LIN {X 0,Y 81.604,Z 314.41,A -85,B 0,C 180,E1 -27784.492,E2 -27784.492} C_VEL
LIN {X 0,Y 79.6,Z 316.274,A -85,B 0,C 180,E1 -27789.318,E2 -27789.318} C_VEL
LIN {X 0,Y 77.196,Z 318.678,A -85,B 0,C 180,E1 -27799.508,E2 -27799.508} C_VEL
LIN {X 0,Y 76.737,Z 319.292,A -85,B 0,C 180,E1 -27804.744,E2 -27804.744} C_VEL
LIN {X 0,Y 76.779,Z 319.509,A -85,B 0,C 180,E1 -27809.999,E2 -27809.999} C_VEL
LIN {X 0,Y 76.737,Z 319.276,A -85,B 0,C 180,E1 -27815.254,E2 -27815.254} C_VEL
LIN {X 0,Y 77.196,Z 318.652,A -85,B 0,C 180,E1 -27820.49,E2 -27820.49} C_VEL
LIN {X 0,Y 78.129,Z 317.638,A -85,B 0,C 180,E1 -27825.655,E2 -27825.655} C_VEL
LIN {X 0,Y 79.599,Z 316.221,A -85,B 0,C 180,E1 -27830.68,E2 -27830.68} C_VEL
LIN {X 0,Y 82.856,Z 313.261,A -85,B 0,C 180,E1 -27837.807,E2 -27837.807} C_VEL
LIN {X 0,Y 87.297,Z 309.266,A -85,B 0,C 180,E1 -27844.3,E2 -27844.3} C_VEL
LIN {X 0,Y 93.773,Z 303.132,A -85,B 0,C 180,E1 -27850.978,E2 -27850.978} C_VEL
LIN {X 0,Y 99.977,Z 296.431,A -85,B 0,C 180,E1 -27856.097,E2 -27856.097} C_VEL
LIN {X 0,Y 104.568,Z 291.112,A -85,B 0,C 180,E1 -27859.121,E2 -27859.121} C_VEL
LIN {X 0,Y 106.383,Z 288.101,A -85,B 0,C 180,E1 -27860.916,E2 -27860.916} C_VEL
LIN {X 0,Y 109.805,Z 280.585,A -85,B 0,C 180,E1 -27865.313,E2 -27865.313} C_VEL
LIN {X 0,Y 110.656,Z 277.96,A -85,B 0,C 180,E1 -27866.879,E2 -27866.879} C_VEL
LIN {X 0,Y 110.746,Z 272.222,A -85,B 0,C 180,E1 -27871.581,E2 -27871.581} C_VEL
LIN {X 0,Y 110.538,Z 266.808,A -85,B 0,C 180,E1 -27876.491,E2 -27876.491} C_VEL
LIN {X 0,Y 110.268,Z 263.922,A -85,B 0,C 180,E1 -27879.479,E2 -27879.479} C_VEL
LIN {X 0,Y 109.572,Z 259.621,A -85,B 0,C 180,E1 -27885.134,E2 -27885.134} C_VEL
LIN {X 0,Y 109.25,Z 257.309,A -85,B 0,C 180,E1 -27888.873,E2 -27888.873} C_VEL
LIN {X 0,Y 108.862,Z 255.868,A -85,B 0,C 180,E1 -27892.582,E2 -27892.582} C_VEL
LIN {X 0,Y 108.806,Z 253.932,A -85,B 0,C 180,E1 -27900,E2 -27900} C_VEL
LIN {X 0,Y 108.95,Z 256.51,A -85,B 0,C 180,E1 -27911.159,E2 -27911.159} C_VEL
LIN {X 0,Y 109.494,Z 258.637,A -85,B 0,C 180,E1 -27915.683,E2 -27915.683} C_VEL
LIN {X 0,Y 110.286,Z 261.526,A -85,B 0,C 180,E1 -27920.517,E2 -27920.517} C_VEL
LIN {X 0,Y 111.3,Z 265.994,A -85,B 0,C 180,E1 -27926.233,E2 -27926.233} C_VEL
LIN {X 0,Y 111.559,Z 271.668,A -85,B 0,C 180,E1 -27931.554,E2 -27931.554} C_VEL
LIN {X 0,Y 111.346,Z 275.635,A -85,B 0,C 180,E1 -27934.863,E2 -27934.863} C_VEL
LIN {X 0,Y 110.502,Z 279.189,A -85,B 0,C 180,E1 -27937.409,E2 -27937.409} C_VEL
LIN {X 0,Y 109.328,Z 282.356,A -85,B 0,C 180,E1 -27939.522,E2 -27939.522} C_VEL
LIN {X 0,Y 102.482,Z 290.942,A -85,B 0,C 180,E1 -27943.942,E2 -27943.942} C_VEL
LIN {X 0,Y 96.019,Z 297.797,A -85,B 0,C 180,E1 -27948.797,E2 -27948.797} C_VEL
LIN {X 0,Y 90.231,Z 303.285,A -85,B 0,C 180,E1 -27954.258,E2 -27954.258} C_VEL
LIN {X 0,Y 85.747,Z 307.295,A -85,B 0,C 180,E1 -27959.943,E2 -27959.943} C_VEL
LIN {X 0,Y 82.984,Z 309.237,A -85,B 0,C 180,E1 -27963.233,E2 -27963.233} C_VEL
LIN {X 0,Y 77.304,Z 311.877,A -85,B 0,C 180,E1 -27968.727,E2 -27968.727} C_VEL
LIN {X 0,Y 73.078,Z 313.418,A -85,B 0,C 180,E1 -27973.741,E2 -27973.741} C_VEL
LIN {X 0,Y 70.958,Z 314.218,A -85,B 0,C 180,E1 -27978.105,E2 -27978.105} C_VEL
LIN {X 0,Y 70.581,Z 314.404,A -85,B 0,C 180,E1 -27979.67,E2 -27979.67} C_VEL
LIN {X 0,Y 69.854,Z 315.108,A -85,B 0,C 180,E1 -27990.001,E2 -27990.001} C_VEL
LIN {X 0,Y 70.791,Z 314.325,A -85,B 0,C 180,E1 -28001.454,E2 -28001.454} C_VEL
LIN {X 0,Y 73.92,Z 312,A -85,B 0,C 180,E1 -28012.354,E2 -28012.354} C_VEL
LIN {X 0,Y 77.737,Z 309.13,A -85,B 0,C 180,E1 -28019.819,E2 -28019.819} C_VEL
LIN {X 0,Y 82.607,Z 305.236,A -85,B 0,C 180,E1 -28026.552,E2 -28026.552} C_VEL
LIN {X 0,Y 88.608,Z 300.204,A -85,B 0,C 180,E1 -28032.392,E2 -28032.392} C_VEL
LIN {X 0,Y 95.28,Z 293.865,A -85,B 0,C 180,E1 -28037.53,E2 -28037.53} C_VEL
LIN {X 0,Y 102.491,Z 285.945,A -85,B 0,C 180,E1 -28042.051,E2 -28042.051} C_VEL
LIN {X 0,Y 103.713,Z 284.466,A -85,B 0,C 180,E1 -28042.771,E2 -28042.771} C_VEL
LIN {X 0,Y 105.478,Z 280.531,A -85,B 0,C 180,E1 -28045.565,E2 -28045.565} C_VEL
LIN {X 0,Y 106.236,Z 276.303,A -85,B 0,C 180,E1 -28049.319,E2 -28049.319} C_VEL
LIN {X 0,Y 106.463,Z 271.152,A -85,B 0,C 180,E1 -28054.59,E2 -28054.59} C_VEL
LIN {X 0,Y 106.236,Z 268.605,A -85,B 0,C 180,E1 -28057.847,E2 -28057.847} C_VEL
LIN {X 0,Y 105.496,Z 264.625,A -85,B 0,C 180,E1 -28064.545,E2 -28064.545} C_VEL
LIN {X 0,Y 105.169,Z 262.927,A -85,B 0,C 180,E1 -28068.435,E2 -28068.435} C_VEL
LIN {X 0,Y 104.899,Z 261.783,A -85,B 0,C 180,E1 -28072.299,E2 -28072.299} C_VEL
LIN {X 0,Y 105.184,Z 260.387,A -85,B 0,C 180,E1 -28080,E2 -28080} C_VEL
LIN {X 0,Y 105.171,Z 262.206,A -85,B 0,C 180,E1 -28087.68,E2 -28087.68} C_VEL
LIN {X 0,Y 105.381,Z 263.849,A -85,B 0,C 180,E1 -28091.541,E2 -28091.541} C_VEL
LIN {X 0,Y 105.599,Z 266.137,A -85,B 0,C 180,E1 -28095.439,E2 -28095.439} C_VEL
LIN {X 0,Y 105.734,Z 269.102,A -85,B 0,C 180,E1 -28099.411,E2 -28099.411} C_VEL
LIN {X 0,Y 105.704,Z 273.818,A -85,B 0,C 180,E1 -28104.554,E2 -28104.554} C_VEL
LIN {X 0,Y 105.345,Z 279.456,A -85,B 0,C 180,E1 -28109.854,E2 -28109.854} C_VEL
LIN {X 0,Y 104.871,Z 281.979,A -85,B 0,C 180,E1 -28111.963,E2 -28111.963} C_VEL
LIN {X 0,Y 101.75,Z 288.088,A -85,B 0,C 180,E1 -28115.748,E2 -28115.748} C_VEL
LIN {X 0,Y 99.967,Z 291.105,A -85,B 0,C 180,E1 -28117.728,E2 -28117.728} C_VEL
LIN {X 0,Y 92.835,Z 298.787,A -85,B 0,C 180,E1 -28122.429,E2 -28122.429} C_VEL
LIN {X 0,Y 85.399,Z 305.878,A -85,B 0,C 180,E1 -28128.823,E2 -28128.823} C_VEL
LIN {X 0,Y 79.781,Z 310.592,A -85,B 0,C 180,E1 -28135.067,E2 -28135.067} C_VEL
LIN {X 0,Y 75.226,Z 314.197,A -85,B 0,C 180,E1 -28142.151,E2 -28142.151} C_VEL
LIN {X 0,Y 72.967,Z 316.06,A -85,B 0,C 180,E1 -28147.338,E2 -28147.338} C_VEL
LIN {X 0,Y 70.207,Z 318.465,A -85,B 0,C 180,E1 -28158.449,E2 -28158.449} C_VEL
LIN {X 0,Y 69.655,Z 319.078,A -85,B 0,C 180,E1 -28164.208,E2 -28164.208} C_VEL
LIN {X 0,Y 69.7,Z 319.297,A -85,B 0,C 180,E1 -28169.999,E2 -28169.999} C_VEL
LIN {X 0,Y 69.654,Z 319.062,A -85,B 0,C 180,E1 -28175.789,E2 -28175.789} C_VEL
LIN {X 0,Y 70.206,Z 318.438,A -85,B 0,C 180,E1 -28181.548,E2 -28181.548} C_VEL
LIN {X 0,Y 71.285,Z 317.424,A -85,B 0,C 180,E1 -28187.202,E2 -28187.202} C_VEL
LIN {X 0,Y 72.966,Z 316.006,A -85,B 0,C 180,E1 -28192.659,E2 -28192.659} C_VEL
LIN {X 0,Y 76.623,Z 313.046,A -85,B 0,C 180,E1 -28200.294,E2 -28200.294} C_VEL
LIN {X 0,Y 81.495,Z 309.05,A -85,B 0,C 180,E1 -28207.131,E2 -28207.131} C_VEL
LIN {X 0,Y 88.486,Z 302.915,A -85,B 0,C 180,E1 -28214.023,E2 -28214.023} C_VEL
LIN {X 0,Y 95.161,Z 296.214,A -85,B 0,C 180,E1 -28219.198,E2 -28219.198} C_VEL
LIN {X 0,Y 99.957,Z 290.891,A -85,B 0,C 180,E1 -28222.276,E2 -28222.276} C_VEL
LIN {X 0,Y 103.637,Z 284.248,A -85,B 0,C 180,E1 -28226.53,E2 -28226.53} C_VEL
LIN {X 0,Y 104.796,Z 281.776,A -85,B 0,C 180,E1 -28228.034,E2 -28228.034} C_VEL
LIN {X 0,Y 105.331,Z 278.155,A -85,B 0,C 180,E1 -28231.127,E2 -28231.127} C_VEL
LIN {X 0,Y 105.641,Z 272.557,A -85,B 0,C 180,E1 -28236.474,E2 -28236.474} C_VEL
LIN {X 0,Y 105.63,Z 268.871,A -85,B 0,C 180,E1 -28240.569,E2 -28240.569} C_VEL
LIN {X 0,Y 105.322,Z 264.758,A -85,B 0,C 180,E1 -28246.494,E2 -28246.494} C_VEL
LIN {X 0,Y 105.259,Z 263.597,A -85,B 0,C 180,E1 -28248.445,E2 -28248.445} C_VEL
LIN {X 0,Y 105.008,Z 262.005,A -85,B 0,C 180,E1 -28252.308,E2 -28252.308} C_VEL
LIN {X 0,Y 105.088,Z 260.062,A -85,B 0,C 180,E1 -28260,E2 -28260} C_VEL
LIN {X 0,Y 104.722,Z 261.568,A -85,B 0,C 180,E1 -28267.714,E2 -28267.714} C_VEL
LIN {X 0,Y 104.988,Z 262.712,A -85,B 0,C 180,E1 -28271.585,E2 -28271.585} C_VEL
LIN {X 0,Y 105.513,Z 265.43,A -85,B 0,C 180,E1 -28277.442,E2 -28277.442} C_VEL
LIN {X 0,Y 106.146,Z 269.313,A -85,B 0,C 180,E1 -28283.408,E2 -28283.408} C_VEL
LIN {X 0,Y 106.325,Z 270.908,A -85,B 0,C 180,E1 -28285.445,E2 -28285.445} C_VEL
LIN {X 0,Y 106.148,Z 275.928,A -85,B 0,C 180,E1 -28290.604,E2 -28290.604} C_VEL
LIN {X 0,Y 105.865,Z 278.277,A -85,B 0,C 180,E1 -28292.819,E2 -28292.819} C_VEL
LIN {X 0,Y 104.975,Z 281.416,A -85,B 0,C 180,E1 -28295.331,E2 -28295.331} C_VEL
LIN {X 0,Y 103.752,Z 284.146,A -85,B 0,C 180,E1 -28297.247,E2 -28297.247} C_VEL
LIN {X 0,Y 96.504,Z 292.383,A -85,B 0,C 180,E1 -28301.716,E2 -28301.716} C_VEL
LIN {X 0,Y 90.803,Z 298.012,A -85,B 0,C 180,E1 -28305.848,E2 -28305.848} C_VEL
LIN {X 0,Y 84.557,Z 303.5,A -85,B 0,C 180,E1 -28311.439,E2 -28311.439} C_VEL
LIN {X 0,Y 79.319,Z 307.8,A -85,B 0,C 180,E1 -28317.886,E2 -28317.886} C_VEL
LIN {X 0,Y 76.38,Z 310.074,A -85,B 0,C 180,E1 -28322.61,E2 -28322.61} C_VEL
LIN {X 0,Y 73.938,Z 311.92,A -85,B 0,C 180,E1 -28327.655,E2 -28327.655} C_VEL
LIN {X 0,Y 70.791,Z 314.284,A -85,B 0,C 180,E1 -28338.549,E2 -28338.549} C_VEL
LIN {X 0,Y 70.581,Z 314.404,A -85,B 0,C 180,E1 -28339.67,E2 -28339.67} C_VEL
